Omron CX-Programmer project 新工程 (CX-Programmer 9.73)

# PLC LHJ_PLC: CQM1H CPU51
; 山东平度光明2003/08/20

## Global symbols (name address type ; comment)
0.00 BOOL  ; 上环升
0.00 BOOL  ; 上环升
0.01 BOOL  ; 上环降
0.01 BOOL  ; 上环降
0.02 BOOL  ; 下环升
0.02 BOOL  ; 下环升
0.03 BOOL  ; 下环降
0.03 BOOL  ; 下环降
0.04 BOOL  ; 支臂进
0.04 BOOL  ; 支臂进
0.05 BOOL  ; 支臂升
0.05 BOOL  ; 支臂升
0.06 BOOL  ; 定型
0.06 BOOL  ; 定型
0.07 BOOL  ; 合模
0.07 BOOL  ; 合模
0.08 BOOL  ; 开模
0.08 BOOL  ; 开模
0.09 BOOL  ; 急停
0.09 BOOL  ; 急停
0.10 BOOL  ; 机械手闭合
0.10 BOOL  ; 机械手闭合
0.11 BOOL  ; 机械手张开
0.11 BOOL  ; 机械手张开
0.12 BOOL  ; 转入
0.12 BOOL  ; 转入
0.13 BOOL  ; 机械手出
0.13 BOOL  ; 机械手出
0.14 BOOL  ; 机械手升
0.14 BOOL  ; 机械手升
0.15 BOOL  ; 机械手降
0.15 BOOL  ; 机械手降
100.00 BOOL  ; 上环升
100.00 BOOL  ; 上环升
100.01 BOOL  ; 上环降
100.01 BOOL  ; 上环降
100.02 BOOL  ; 下环升
100.02 BOOL  ; 下环升
100.03 BOOL  ; 下环降
100.03 BOOL  ; 下环降
100.04 BOOL  ; 支臂进
100.04 BOOL  ; 支臂进
100.05 BOOL  ; 支臂出
100.05 BOOL  ; 支臂出
100.06 BOOL  ; 支臂停
100.06 BOOL  ; 支臂停
100.07 BOOL  ; 支臂升
100.07 BOOL  ; 支臂升
100.08 BOOL  ; 油泵进
100.08 BOOL  ; 油泵进
100.09 BOOL  ; 油泵回
100.09 BOOL  ; 油泵回
100.10 BOOL  ; 合模换向
100.10 BOOL  ; 合模换向
100.11 BOOL  ; 开模换向
100.11 BOOL  ; 开模换向
100.12 BOOL  ; 抱闸
100.12 BOOL  ; 抱闸
100.13 BOOL  ; 合模
100.13 BOOL  ; 合模
100.14 BOOL  ; 开模
100.14 BOOL  ; 开模
101.00 BOOL  ; 定型
101.00 BOOL  ; 定型
101.01 BOOL  ; 二次定型
101.01 BOOL  ; 二次定型
101.02 BOOL  ; 左手闭合
101.02 BOOL  ; 左手闭合
101.03 BOOL  ; 右手闭合
101.03 BOOL  ; 右手闭合
101.04 BOOL  ; 左手降
101.04 BOOL  ; 左手降
101.05 BOOL  ; 右手降
101.05 BOOL  ; 右手降
101.06 BOOL  ; 左手停
101.06 BOOL  ; 左手停
101.07 BOOL  ; 右手停
101.07 BOOL  ; 右手停
101.08 BOOL  ; 左手入
101.08 BOOL  ; 左手入
101.09 BOOL  ; 右手入
101.09 BOOL  ; 右手入
101.10 BOOL  ; 左手出
101.10 BOOL  ; 左手出
101.11 BOOL  ; 右手出
101.11 BOOL  ; 右手出
101.12 BOOL  ; 自动指示灯
101.12 BOOL  ; 自动指示灯
101.13 BOOL  ; 硫化压力灯
101.14 BOOL  ; 硫化压力灯
101.14 BOOL  ; 硫化灯
101.15 BOOL  ; 硫化，延时硫化灯
101.15 BOOL  ; 硫化，延时硫化灯
102.00 BOOL  ; 内压蒸汽进
102.00 BOOL  ; 内压蒸汽进
102.01 BOOL  ; 内压蒸汽关
102.01 BOOL  ; 内压蒸汽关
102.02 BOOL  ; 二次水开
102.02 BOOL  ; 二次水开
102.03 BOOL  ; 二次水关
102.03 BOOL  ; 二次水关
102.04 BOOL  ; 热水回开
102.04 BOOL  ; 热水回开
102.05 BOOL  ; 热水回关
102.05 BOOL  ; 热水回关
102.06 BOOL  ; 5BAR热水回开
102.06 BOOL  ; 5BAR热水回开
102.07 BOOL  ; 5BAR热水回关
102.07 BOOL  ; 5BAR热水回关
102.08 BOOL  ; 0BAR热水回开
102.08 BOOL  ; 0BAR热水回开
102.09 BOOL  ; 0BAR热水回关
102.09 BOOL  ; 0BAR热水回关
102.10 BOOL  ; 抽真空开
102.11 BOOL  ; 抽真空关
102.12 BOOL  ; 外压（温）进开
102.13 BOOL  ; 外压（温）进关
102.14 BOOL  ; 冷水进回开
102.14 BOOL  ; 冷水进回开
102.15 BOOL  ; 冷水进回关
102.15 BOOL  ; 冷水进回关
103.00 BOOL  ; 外温进开
103.00 BOOL  ; 外温进开
103.01 BOOL  ; 活络模缩
103.02 BOOL  ; 活络模伸
103.02 BOOL  ; 活络模伸
103.03 BOOL  ; 活络模缩
103.03 BOOL  ; 活络模缩
103.04 BOOL  ; 挡胎杆降
103.04 BOOL  ; 挡胎杆降
103.05 BOOL  ; 活络模溢流
103.06 BOOL  ; 下环降停阀（有电通水）
103.08 BOOL  ; 报警灯
103.10 BOOL  ; 正常状态灯
103.12 BOOL  ; 程控气源失压报警
103.12 BOOL  ; 程控气源失压报警
104 CHANNEL  ; 外温回汽
104 CHANNEL  ; 外温回汽
105 CHANNEL  ; 进汽
105 CHANNEL  ; 进汽
11.10 BOOL  ; 左手转出
11.10 BOOL  ; 左手转出
13.15 BOOL  ; 延时硫化信号
13.15 BOOL  ; 延时硫化信号
14.00 BOOL  ; 实际压力大于设定的0.5公斤
14.00 BOOL  ; 实际压力大于设定的0.5公斤
15.00 BOOL  ; 备用
15.05 BOOL  ; 13.13
1.00 BOOL  ; 机械手停
1.00 BOOL  ; 机械手停
1.01 BOOL  ; 硫化延时
1.01 BOOL  ; 硫化延时
1.04 BOOL  ; 程序控制器
1.04 BOOL  ; 程序控制器
1.05 BOOL  ; 自动
1.05 BOOL  ; 自动
1.06 BOOL  ; 手动排
1.06 BOOL  ; 手动排
1.07 BOOL  ; 润滑
1.07 BOOL  ; 润滑
1.08 BOOL  ; 返回
1.08 BOOL  ; 返回
1.09 BOOL  ; 活络模升
1.09 BOOL  ; 活络模伸
1.10 BOOL  ; 活络模缩
1.10 BOOL  ; 活络模缩
1.11 BOOL  ; 挡胎杆升
1.13 BOOL  ; 机手（左）
1.13 BOOL  ; 机手（左）
1.14 BOOL  ; 机械手双
1.14 BOOL  ; 机械手双
1.15 BOOL  ; 机手（右）
1.15 BOOL  ; 机手（右）
22 CHANNEL  ; 动作序号
22.00 BOOL  ; 开模极限（编）
22.00 BOOL  ; 开模极限（编）
22.01 BOOL  ; 下环升
22.01 BOOL  ; 下环升
22.02 BOOL  ; 合模停（编）
22.02 BOOL  ; 合模停（编）
22.03 BOOL  ; 二次定型（编）
22.03 BOOL  ; 二次定型（编）
22.04 BOOL  ; 合模极限（编）
22.04 BOOL  ; 合模极限（编）
22.05 BOOL  ; 活络模伸（编）
22.05 BOOL  ; 活络模伸（编）
22.06 BOOL  ; 活络模缩（编）
22.06 BOOL  ; 活络模缩（编）
22.07 BOOL  ; 活络模保持
22.07 BOOL  ; 活络模保持
22 CHANNEL  ; 动作序号
233 CHANNEL  ; 热板温度采集
234 CHANNEL  ; 模套温度采集
236 CHANNEL  ; 模套温度电气转换器控制值
237 CHANNEL  ; 热板温度电气转换器控制值
23.00 BOOL  ; 达到设定步序
23.00 BOOL  ; 达到设定步序
26 CHANNEL  ; 判断步时间设定为0
26.00 BOOL  ; 第1步时间为0
26.00 BOOL  ; 第1步时间为0
26.01 BOOL  ; 第2步时间为0
26.01 BOOL  ; 第2步时间为0
26.02 BOOL  ; 第3步时间为0
26.02 BOOL  ; 第3步时间为0
26.03 BOOL  ; 第4步时间为0
26.03 BOOL  ; 第4步时间为0
26.04 BOOL  ; 第5步时间为0
26.04 BOOL  ; 第5步时间为0
26.05 BOOL  ; 第6步时间为0
26.05 BOOL  ; 第6步时间为0
26.06 BOOL  ; 第7步时间为0
26.06 BOOL  ; 第7步时间为0
26.07 BOOL  ; 8步时间为0
26.07 BOOL  ; 8步时间为0
26.08 BOOL  ; 九步时间为0
26.08 BOOL  ; 九步时间为0
26.09 BOOL  ; 第十步时间为0
26.09 BOOL  ; 第十步时间为0
26.10 BOOL  ; 11步时间为0
26.10 BOOL  ; 11步时间为0
26.11 BOOL  ; 12步时间为0
26.11 BOOL  ; 12步时间为0
26.12 BOOL  ; 第13步时间为0
26.12 BOOL  ; 第13步时间为0
26.13 BOOL  ; 第14步时间为0
26.13 BOOL  ; 第14步时间为0
26.14 BOOL  ; 第15步时间为0
26.14 BOOL  ; 第15步时间为0
26.15 BOOL  ; 第16步时间为0
26.15 BOOL  ; 第16步时间为0
26 CHANNEL  ; 判断步时间设定为0
2.00 BOOL  ; 抱闸
2.00 BOOL  ; 抱闸
2.01 BOOL  ; 内压
2.03 BOOL  ; 下环升
2.03 BOOL  ; 下环升
2.04 BOOL  ; 下环降
2.04 BOOL  ; 下环降
2.05 BOOL  ; 支臂进
2.05 BOOL  ; 支臂进
2.06 BOOL  ; 支臂停
2.06 BOOL  ; 支臂停
2.07 BOOL  ; 支臂降
2.07 BOOL  ; 支臂降
2.08 BOOL  ; 支臂出
2.08 BOOL  ; 支臂出
2.09 BOOL  ; 左手张开
2.09 BOOL  ; 左手张开
2.10 BOOL  ; 右手张开
2.10 BOOL  ; 右手张开
2.11 BOOL  ; 左手闭合
2.11 BOOL  ; 左手闭合
2.12 BOOL  ; 右手闭合
2.12 BOOL  ; 右手闭合
2.15 BOOL  ; 左手上限
2.15 BOOL  ; 左手上限
30.00 BOOL  ; 安全联锁
30.00 BOOL  ; 安全联锁
30.01 BOOL  ; 下环联锁
30.01 BOOL  ; 下环联锁
30.02 BOOL  ; 支臂联锁
30.02 BOOL  ; 支臂联锁
30.03 BOOL  ; 机手联锁
30.03 BOOL  ; 机手联锁
30.15 BOOL  ; 动作条件
30.15 BOOL  ; 动作条件
3.00 BOOL  ; 右手上限
3.00 BOOL  ; 右手上限
3.01 BOOL  ; 左手入
3.01 BOOL  ; 左手入
3.02 BOOL  ; 右手入
3.02 BOOL  ; 右手入
3.03 BOOL  ; 左手转出
3.03 BOOL  ; 左手转出
3.04 BOOL  ; 右手转出
3.04 BOOL  ; 右手转出
3.05 BOOL  ; 左手放胎
3.05 BOOL  ; 左手放胎
3.06 BOOL  ; 右手放胎
3.06 BOOL  ; 右手放胎
3.07 BOOL  ; 左手触胎
3.07 BOOL  ; 左手触胎
3.08 BOOL  ; 右手触胎
3.08 BOOL  ; 右手触胎
3.09 BOOL  ; 合模极限
3.09 BOOL  ; 合模极限
3.10 BOOL  ; 开模极限
3.10 BOOL  ; 开模极限
3.11 BOOL  ; 左安全开关
3.11 BOOL  ; 左安全开关
3.12 BOOL  ; 右安全开关
3.12 BOOL  ; 右安全开关
3.13 BOOL  ; 左活络模伸
3.13 BOOL  ; 左活络模伸
3.14 BOOL  ; 右活络模伸
3.14 BOOL  ; 右活络模伸
3.15 BOOL  ; 左活络模缩
3.15 BOOL  ; 左活络模缩
40.05 BOOL  ; 自动合模
40.05 BOOL  ; 自动合模
40.06 BOOL  ; 合模延时自锁
40.06 BOOL  ; 合模延时自锁
40.07 BOOL  ; 合模
40.07 BOOL  ; 合模
40.10 BOOL  ; 开模条件
40.10 BOOL  ; 开模条件
40.11 BOOL  ; 开模
40.11 BOOL  ; 开模
40.12 BOOL  ; 上环升条件1
40.12 BOOL  ; 上环升条件1
40.13 BOOL  ; 上环升条件1+2
40.13 BOOL  ; 上环升条件1+2
40.14 BOOL  ; 下环升条件
40.14 BOOL  ; 下环升条件
40.15 BOOL  ; 卸胎支臂停条件
40.15 BOOL  ; 卸胎支臂停条件
41.01 BOOL  ; 下环升
41.01 BOOL  ; 下环升
42.15 BOOL  ; 自动
42.15 BOOL  ; 自动
49.07 BOOL  ; 8-16步时间
49.07 BOOL  ; 8-16步时间
49.13 BOOL  ; 硫化结束步序清零
49.13 BOOL  ; 硫化结束步序清零
49.14 BOOL  ; 硫化结束
49.14 BOOL  ; 硫化结束
4.00 BOOL  ; 右活络模缩
4.00 BOOL  ; 右活络模缩
4.01 BOOL  ; 编码器输入1
4.01 BOOL  ; 编码器输入1
4.02 BOOL  ; 编码器输入2
4.02 BOOL  ; 编码器输入2
4.03 BOOL  ; 编码器输入3
4.03 BOOL  ; 编码器输入3
4.04 BOOL  ; 编码器输入4
4.04 BOOL  ; 编码器输入4
4.05 BOOL  ; 编码器输入5
4.05 BOOL  ; 编码器输入5
4.06 BOOL  ; 编码器输入6
4.06 BOOL  ; 编码器输入6
4.07 BOOL  ; 编码器输入7
4.07 BOOL  ; 编码器输入7
4.08 BOOL  ; 编码器输入8
4.08 BOOL  ; 编码器输入8
4.11 BOOL  ; 机械手切换
4.11 BOOL  ; 机械手切换
5 CHANNEL  ; 外温码
50.00 BOOL  ; 机械手转入自动
50.00 BOOL  ; 机械手转入自动
50.01 BOOL  ; 机械手转入自动
50.01 BOOL  ; 机械手转入自动
50.02 BOOL  ; 机手放胎条件
50.02 BOOL  ; 机手放胎条件
50.04 BOOL  ; 机手入自锁
50.04 BOOL  ; 机手入自锁
51.00 BOOL  ; 合模信号
51.00 BOOL  ; 合模信号
59.15 BOOL  ; 硫化条件
59.15 BOOL  ; 硫化条件
5 CHANNEL  ; 外温码
75.00 BOOL  ; 15步走完脉冲
75.00 BOOL  ; 15步走完脉冲
75.02 BOOL  ; 1步走完脉冲
75.02 BOOL  ; 1步走完脉冲
75.03 BOOL  ; 2步走完脉冲
75.03 BOOL  ; 2步走完脉冲
75.15 BOOL  ; 14步走完脉冲
75.15 BOOL  ; 14步走完脉冲
76.00 BOOL  ; 16步走完脉冲
76.00 BOOL  ; 16步走完脉冲
79.00 BOOL  ; 左闭合信号
79.00 BOOL  ; 左闭合信号
79.01 BOOL  ; 右闭信号
79.01 BOOL  ; 右闭信号
CNT001 BOOL  ; 初始化
CNT001 BOOL  ; 初始化
CNT002 BOOL  ; 第一步时间
CNT002 BOOL  ; 第一步时间
CNT003 BOOL  ; 第二步时间
CNT003 BOOL  ; 第二步时间
CNT004 BOOL  ; 第三步时间
CNT004 BOOL  ; 第三步时间
CNT005 BOOL  ; 第4步时间
CNT005 BOOL  ; 第4步时间
CNT006 BOOL  ; 第五步时间
CNT006 BOOL  ; 第五步时间
CNT007 BOOL  ; 第6步时间
CNT007 BOOL  ; 第6步时间
CNT008 BOOL  ; 第7步时间
CNT008 BOOL  ; 第7步时间
CNT009 BOOL  ; 第八步时
CNT009 BOOL  ; 第八步时
CNT010 BOOL  ; 第九步时
CNT010 BOOL  ; 第九步时
CNT011 BOOL  ; 第十步时
CNT011 BOOL  ; 第十步时
CNT012 BOOL  ; 第11步时间
CNT012 BOOL  ; 第11步时间
CNT013 BOOL  ; 第12步时间
CNT013 BOOL  ; 第12步时间
CNT014 BOOL  ; 第13步时间
CNT014 BOOL  ; 第13步时间
CNT015 BOOL  ; 第14步时间
CNT015 BOOL  ; 第14步时间
CNT016 BOOL  ; 第15步时间
CNT016 BOOL  ; 第15步时间
CNT017 BOOL  ; 第16步时间
CNT017 BOOL  ; 第16步时间
CNT018 BOOL  ; 硫化复位
CNT018 BOOL  ; 硫化复位
CNT022 BOOL  ; 延时硫化时间
CNT022 BOOL  ; 延时硫化时间
DM10 CHANNEL  ; 硫化总时间
DM1020 CHANNEL  ; PID模套温度设定二进值码
DM1021 CHANNEL  ; PID模套温度P参数
DM1026 CHANNEL  ; 模套温度PID的C+6
DM1055 CHANNEL  ; 模套温度PID控回汽
DM1055 CHANNEL  ; 温度PID控回汽
DM1060 CHANNEL  ; PID热板设定二进制码
DM1061 CHANNEL  ; PID热板P参数
DM1066 CHANNEL  ; 热板PID的C+6
DM1120 CHANNEL  ; 模套实际显示值
DM1122 CHANNEL  ; 内温实际显示值
DM1122 CHANNEL  ; 内温实际显示值
DM1126 CHANNEL  ; 内压实际显示值
DM1126 CHANNEL  ; 内压实际显示值
DM1128 CHANNEL  ; 实际热板温度显示值
DM1148 CHANNEL  ; 设定值加0.05公斤
DM1148 CHANNEL  ; 设定值加0.05公斤
DM1207 CHANNEL  ; 模套温度PID控制
DM1212 CHANNEL  ; 热板温度PID控制
DM1214 CHANNEL  ; 进汽阀开启度
DM1214 CHANNEL  ; 模套进汽阀开启度
DM1220 CHANNEL  ; 模套实际外温二进值码
DM1222 CHANNEL  ; 实际内温二进制码
DM1222 CHANNEL  ; 实际内温二进制码
DM1224 CHANNEL  ; 实际内压二进制码
DM1224 CHANNEL  ; 实际内压二进制码
DM1226 CHANNEL  ; 实际外压二进制码
DM1226 CHANNEL  ; 实际外压二进制码
DM1228 CHANNEL  ; PID热板实际温度二进值码
DM1230 CHANNEL  ; 实际内压MPa
DM1230 CHANNEL  ; 实际内压MPa
DM1232 CHANNEL  ; 实际外压MPa
DM1232 CHANNEL  ; 实际外压MPa
DM1238 CHANNEL  ; 压力低于设定值0.1公斤
DM1238 CHANNEL  ; 压力低于设定值0.1公斤
DM1242 CHANNEL  ; 热板进汽阀门开启度
DM170 CHANNEL  ; 模套温度设定值二进值码
DM172 CHANNEL  ; PPC热板温度设定值二进值码
DM400 CHANNEL  ; 步序一时间
DM400 CHANNEL  ; 步序一时间
DM401 CHANNEL  ; 步序二时间
DM401 CHANNEL  ; 步序二时间
DM402 CHANNEL  ; 步序三时间
DM402 CHANNEL  ; 步序三时间
DM403 CHANNEL  ; 步序四时间
DM403 CHANNEL  ; 步序四时间
DM404 CHANNEL  ; 步序五时间
DM404 CHANNEL  ; 步序五时间
DM405 CHANNEL  ; 步序六时间
DM405 CHANNEL  ; 步序六时间
DM406 CHANNEL  ; 步序七时间
DM406 CHANNEL  ; 步序七时间
DM407 CHANNEL  ; 第八步时间
DM407 CHANNEL  ; 第八步时间
DM408 CHANNEL  ; 第九步时间
DM408 CHANNEL  ; 第九步时间
DM409 CHANNEL  ; 第十步时间
DM409 CHANNEL  ; 第十步时间
DM410 CHANNEL  ; 第11步时间
DM410 CHANNEL  ; 第11步时间
DM411 CHANNEL  ; 第12步时间
DM411 CHANNEL  ; 第12步时间
DM412 CHANNEL  ; 第13步时间
DM412 CHANNEL  ; 第13步时间
DM413 CHANNEL  ; 第14步时间
DM413 CHANNEL  ; 第14步时间
DM414 CHANNEL  ; 第15步时间
DM414 CHANNEL  ; 第15步时间
DM415 CHANNEL  ; 第16步时间
DM415 CHANNEL  ; 第16步时间
DM416 CHANNEL  ; 第1步阀门状态
DM416 CHANNEL  ; 第1步阀门状态
DM417 CHANNEL  ; 第2步阀门状态
DM417 CHANNEL  ; 第2步阀门状态
DM418 CHANNEL  ; 第3步阀门状态
DM418 CHANNEL  ; 第3步阀门状态
DM419 CHANNEL  ; 第4步阀门状态
DM419 CHANNEL  ; 第4步阀门状态
DM420 CHANNEL  ; 第5步阀门状态
DM420 CHANNEL  ; 第5步阀门状态
DM421 CHANNEL  ; 第6步阀门状态
DM421 CHANNEL  ; 第6步阀门状态
DM422 CHANNEL  ; 第7步阀门状态
DM422 CHANNEL  ; 第7步阀门状态
DM423 CHANNEL  ; 第8步 阀门状态
DM423 CHANNEL  ; 第8步 阀门状态
DM424 CHANNEL  ; 第9步阀门状态
DM424 CHANNEL  ; 第9步阀门状态
DM425 CHANNEL  ; 第10步阀门状态
DM425 CHANNEL  ; 第10步阀门状态
DM426 CHANNEL  ; 第11步阀门状态
DM426 CHANNEL  ; 第11步阀门状态
DM427 CHANNEL  ; 第12步阀门状态
DM427 CHANNEL  ; 第12步阀门状态
DM428 CHANNEL  ; 第13步阀门状态
DM428 CHANNEL  ; 第13步阀门状态
DM429 CHANNEL  ; 第14步阀门状态
DM429 CHANNEL  ; 第14步阀门状态
DM430 CHANNEL  ; 第15步阀门状态
DM430 CHANNEL  ; 第15步阀门状态
DM431 CHANNEL  ; 第16步阀门状态
DM431 CHANNEL  ; 第16步阀门状态
DM448 CHANNEL  ; 模套设定值
DM449 CHANNEL  ; PPC写模套P参数
DM460 CHANNEL  ; PPC写热板温度设定值
DM461 CHANNEL  ; PPC写热板P参数
DM489 CHANNEL  ; 合模延时时间
DM489 CHANNEL  ; 合模延时时间
DM490 CHANNEL  ; 卸胎臂停延时
DM490 CHANNEL  ; 卸胎臂停延时
DM491 CHANNEL  ; 机械手闭合延时
DM491 CHANNEL  ; 机械手闭合延时
DM492 CHANNEL  ; 上环降延时
DM492 CHANNEL  ; 上环降延时
DM495 CHANNEL  ; 上环升延时
DM495 CHANNEL  ; 下环降延时
DM496 CHANNEL  ; 硫化延时时间
DM496 CHANNEL  ; 硫化延时时间
DM503 CHANNEL  ; 总步序设定
DM503 CHANNEL  ; 总步序设定
DM800 CHANNEL  ; 位置表比较
DM800 CHANNEL  ; 位置表比较
DM930 CHANNEL  ; PPC读PLC外温二进制数
DM930 CHANNEL  ; PPC读PLC外温二进制数
DM931 CHANNEL  ; PPC读PLC内温二进制数
DM931 CHANNEL  ; PPC读PLC内温二进制数
DM932 CHANNEL  ; PPC读PLC内压二进制数
DM932 CHANNEL  ; PPC读PLC内压二进制数
DM933 CHANNEL  ; PPC读PLC外压二进制数
DM933 CHANNEL  ; PPC读PLC外压二进制数
DM934 CHANNEL  ; 硫化总时间显示
DM934 CHANNEL  ; 硫化总时间显示
DM935 CHANNEL  ; 步序时间显示
DM935 CHANNEL  ; 步序时间显示
DM936 CHANNEL  ; PPC硫化延时显示
DM936 CHANNEL  ; PPC硫化延时显示
DM937 CHANNEL  ; 模套进汽阀开启度
DM937 CHANNEL  ; 进汽阀开启度
DM938 CHANNEL  ; 编码器值
DM938 CHANNEL  ; 编码器值
DM939 CHANNEL  ; 当前步序
DM939 CHANNEL  ; 当前步序
DM940 CHANNEL  ; 总剩余时间
DM940 CHANNEL  ; 总剩余时间
DM941 CHANNEL  ; 阀门状态
DM941 CHANNEL  ; 阀门状态
DM942 CHANNEL  ; 硫化状态标志
DM942 CHANNEL  ; 硫化状态标志
DM943 CHANNEL  ; PPC读00-01通道地址
DM943 CHANNEL  ; PPC读00-01通道地址
DM945 CHANNEL  ; PPC读PLC02-03通道地址
DM945 CHANNEL  ; PPC读PLC02-03通道地址
DM947 CHANNEL  ; PPC读100-103通道地址
DM947 CHANNEL  ; PPC读100-103通道地址
DM951 CHANNEL  ; PPC热板进汽阀门开启度
HR31.00 BOOL  ; 自动硫化保护
HR31.00 BOOL  ; 自动硫化保护
TIM000 BOOL  ; 合模延时时间
TIM000 BOOL  ; 合模延时时间
TIM052 BOOL  ; 下环降延时
TIM052 BOOL  ; 下环降延时
TIM053 BOOL  ; 卸胎支臂停延时
TIM053 BOOL  ; 卸胎支臂停延时
TIM054 BOOL  ; 上环降延时
TIM054 BOOL  ; 上环降延时
TIM056 BOOL  ; 返回时间
TIM056 BOOL  ; 返回时间
TIM057 BOOL  ; 润滑时间
TIM057 BOOL  ; 润滑时间
TIM069 BOOL  ; 支臂降延时
TIM069 BOOL  ; 支臂降延时
TIM070 BOOL  ; 定型延时
TIM070 BOOL  ; 机械手闭合延时
TIM071 BOOL  ; 左手在外抓胎延时
TIM071 BOOL  ; 左手在外抓胎延时
TIM072 BOOL  ; 右手在外抓胎延时
TIM072 BOOL  ; 右手在外抓胎延时
TIM079 BOOL  ; 内压
TIM079 BOOL  ; 内压

## Program 新程序1 (no task)
; 系统使用欧姆龙PLC CQM1H CPU51，通过编码器、温度传感器、压力传感器、机械手、阀门和安全开关等设备实现硫化过程的自动化控制。 / 系统只有在急停未触发且安全门关闭时，硫化流程才会启动，否则所有动作如合模和开模立即停止，确保操作安全。 / 硫化过程温度控制通过PID算法实现，利用PID模套温度设定值和PID热板温度设定值调整模套温度控制值和热板温度控制值，使温度稳定在设定值的±5%以内，确保硫化质量。 / 压力则通过内压蒸汽进和内压蒸汽关调节，保持在设定值的±0.5巴范围内，避免压力波动影响轮胎成型。 / 机械手动作由左手闭合、右手闭合、左手入、右手入等信号驱动，且左手闭合和右手闭合不会同时激活，且只能在编码器确认的安全区域内执行，防止机械冲突和越界。 / 硫化结束后，计时器触发复位，自动指示灯和硫化灯显示运行状态，系统准备下一轮操作。 / sn:3911-5900-9079-9900

### Section 段1

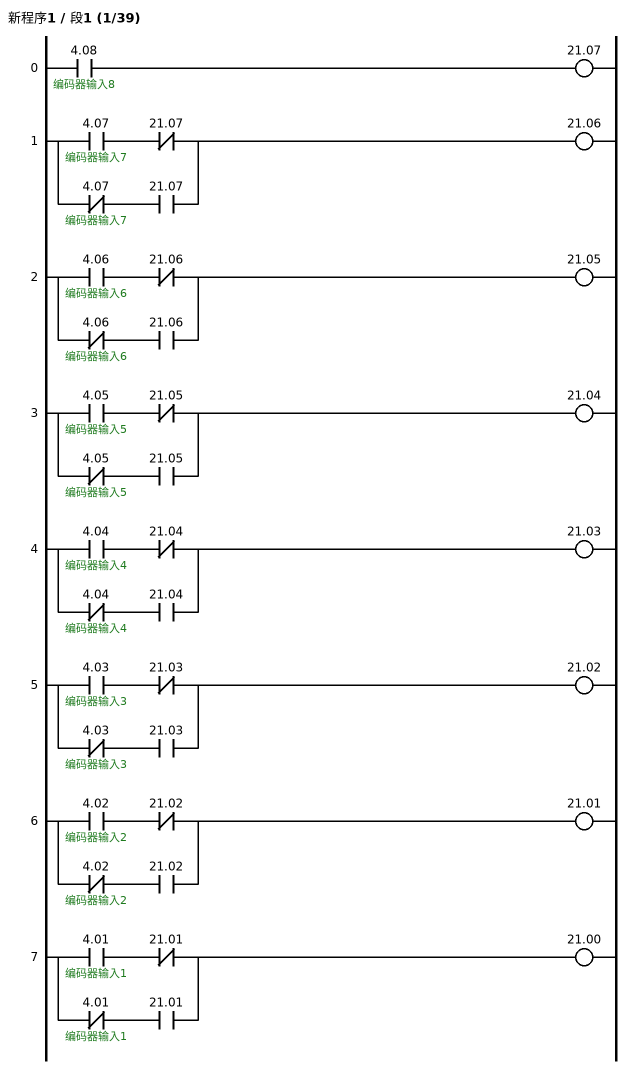
; rung 0
LD 4.08  ; 编码器输入8
OUT 21.07
; rung 1
LD 4.07  ; 编码器输入7
ANDNOT 21.07
LDNOT 4.07  ; 编码器输入7
AND 21.07
ORLD
OUT 21.06
; rung 2
LD 4.06  ; 编码器输入6
ANDNOT 21.06
LDNOT 4.06  ; 编码器输入6
AND 21.06
ORLD
OUT 21.05
; rung 3
LD 4.05  ; 编码器输入5
ANDNOT 21.05
LDNOT 4.05  ; 编码器输入5
AND 21.05
ORLD
OUT 21.04
; rung 4
LD 4.04  ; 编码器输入4
ANDNOT 21.04
LDNOT 4.04  ; 编码器输入4
AND 21.04
ORLD
OUT 21.03
; rung 5
LD 4.03  ; 编码器输入3
ANDNOT 21.03
LDNOT 4.03  ; 编码器输入3
AND 21.03
ORLD
OUT 21.02
; rung 6
LD 4.02  ; 编码器输入2
ANDNOT 21.02
LDNOT 4.02  ; 编码器输入2
AND 21.02
ORLD
OUT 21.01
; rung 7
LD 4.01  ; 编码器输入1
ANDNOT 21.01
LDNOT 4.01  ; 编码器输入1
AND 21.01
ORLD
OUT 21.00

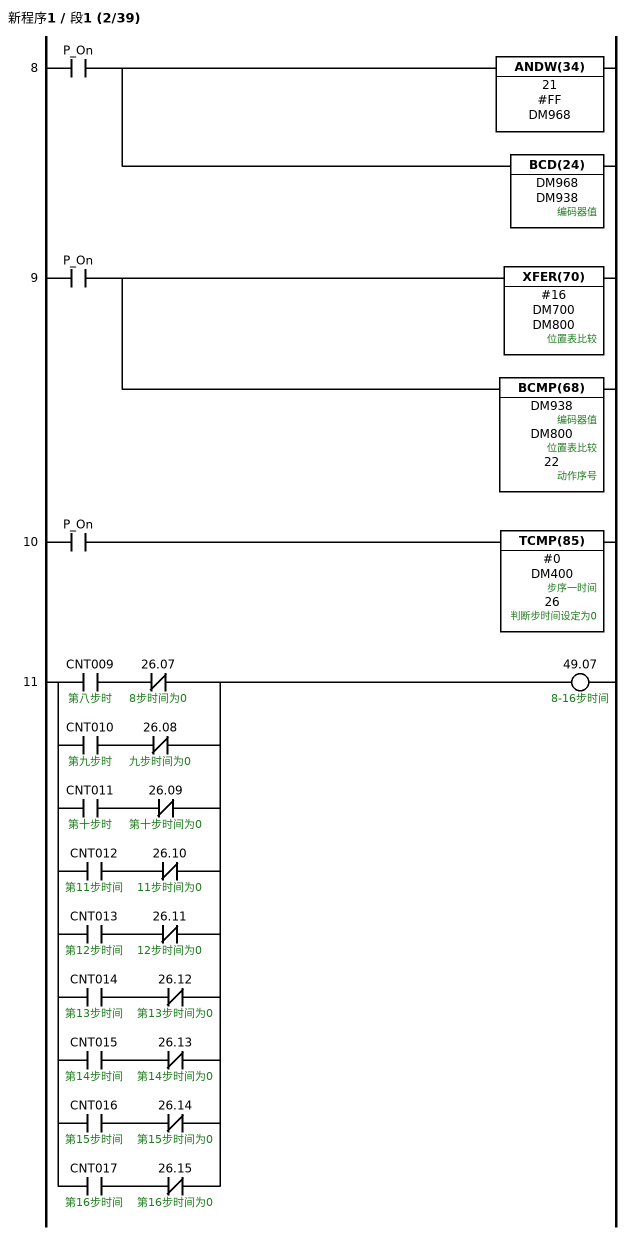
; rung 8
LD P_On
ANDW(34) 21 #FF DM968
BCD(24) DM968 DM938  ; 编码器值
; rung 9
LD P_On
XFER(70) #16 DM700 DM800  ; 位置表比较
BCMP(68) DM938 DM800 22  ; 编码器值, 位置表比较, 动作序号
; rung 10
LD P_On
TCMP(85) #0 DM400 26  ; 步序一时间, 判断步时间设定为0
; rung 11
LD CNT009  ; 第八步时
ANDNOT 26.07  ; 8步时间为0
LD CNT010  ; 第九步时
ANDNOT 26.08  ; 九步时间为0
ORLD
LD CNT011  ; 第十步时
ANDNOT 26.09  ; 第十步时间为0
ORLD
LD CNT012  ; 第11步时间
ANDNOT 26.10  ; 11步时间为0
ORLD
LD CNT013  ; 第12步时间
ANDNOT 26.11  ; 12步时间为0
ORLD
LD CNT014  ; 第13步时间
ANDNOT 26.12  ; 第13步时间为0
ORLD
LD CNT015  ; 第14步时间
ANDNOT 26.13  ; 第14步时间为0
ORLD
LD CNT016  ; 第15步时间
ANDNOT 26.14  ; 第15步时间为0
ORLD
LD CNT017  ; 第16步时间
ANDNOT 26.15  ; 第16步时间为0
ORLD
OUT 49.07  ; 8-16步时间

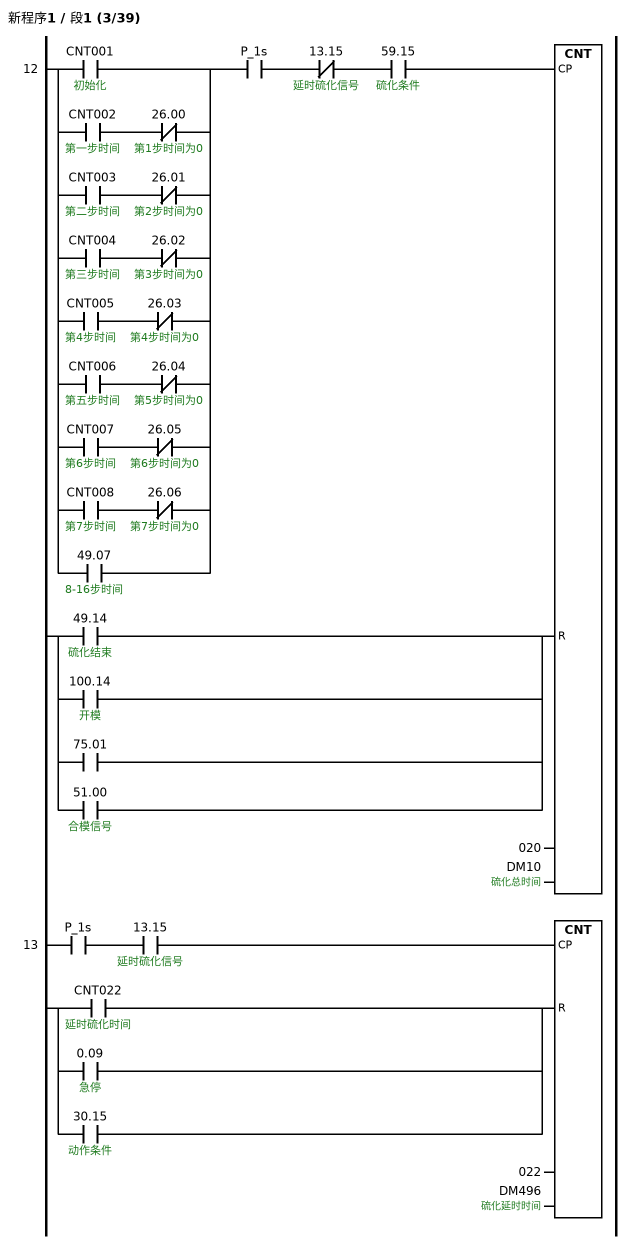
; rung 12
LD CNT001  ; 初始化
LD CNT002  ; 第一步时间
ANDNOT 26.00  ; 第1步时间为0
ORLD
LD CNT003  ; 第二步时间
ANDNOT 26.01  ; 第2步时间为0
ORLD
LD CNT004  ; 第三步时间
ANDNOT 26.02  ; 第3步时间为0
ORLD
LD CNT005  ; 第4步时间
ANDNOT 26.03  ; 第4步时间为0
ORLD
LD CNT006  ; 第五步时间
ANDNOT 26.04  ; 第5步时间为0
ORLD
LD CNT007  ; 第6步时间
ANDNOT 26.05  ; 第6步时间为0
ORLD
LD CNT008  ; 第7步时间
ANDNOT 26.06  ; 第7步时间为0
ORLD
OR 49.07  ; 8-16步时间
AND P_1s
ANDNOT 13.15  ; 延时硫化信号
AND 59.15  ; 硫化条件
LD 49.14  ; 硫化结束
OR 100.14  ; 开模
OR 75.01
OR 51.00  ; 合模信号
CNT 020 DM10  ; 硫化总时间
; rung 13
LD P_1s
AND 13.15  ; 延时硫化信号
LD CNT022  ; 延时硫化时间
OR 0.09  ; 急停
OR 30.15  ; 动作条件
CNT 022 DM496  ; 硫化延时时间

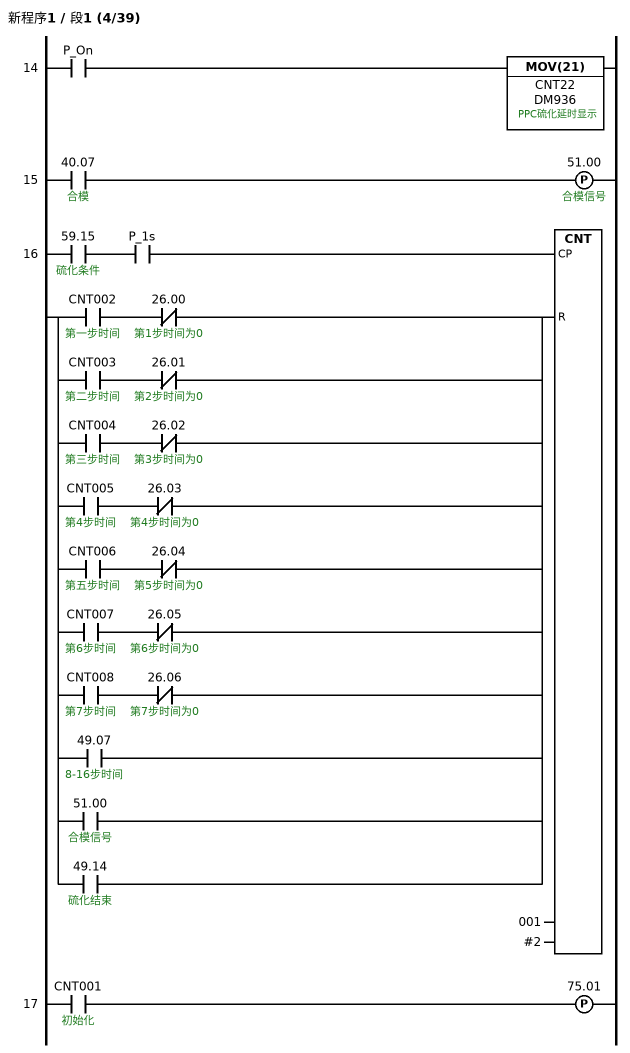
; rung 14
LD P_On
MOV(21) CNT22 DM936  ; PPC硫化延时显示
; rung 15
LD 40.07  ; 合模
DIFU(13) 51.00  ; 合模信号
; rung 16
LD 59.15  ; 硫化条件
AND P_1s
LD CNT002  ; 第一步时间
ANDNOT 26.00  ; 第1步时间为0
LD CNT003  ; 第二步时间
ANDNOT 26.01  ; 第2步时间为0
ORLD
LD CNT004  ; 第三步时间
ANDNOT 26.02  ; 第3步时间为0
ORLD
LD CNT005  ; 第4步时间
ANDNOT 26.03  ; 第4步时间为0
ORLD
LD CNT006  ; 第五步时间
ANDNOT 26.04  ; 第5步时间为0
ORLD
LD CNT007  ; 第6步时间
ANDNOT 26.05  ; 第6步时间为0
ORLD
LD CNT008  ; 第7步时间
ANDNOT 26.06  ; 第7步时间为0
ORLD
OR 49.07  ; 8-16步时间
OR 51.00  ; 合模信号
OR 49.14  ; 硫化结束
CNT 001 #2
; rung 17
LD CNT001  ; 初始化
DIFU(13) 75.01

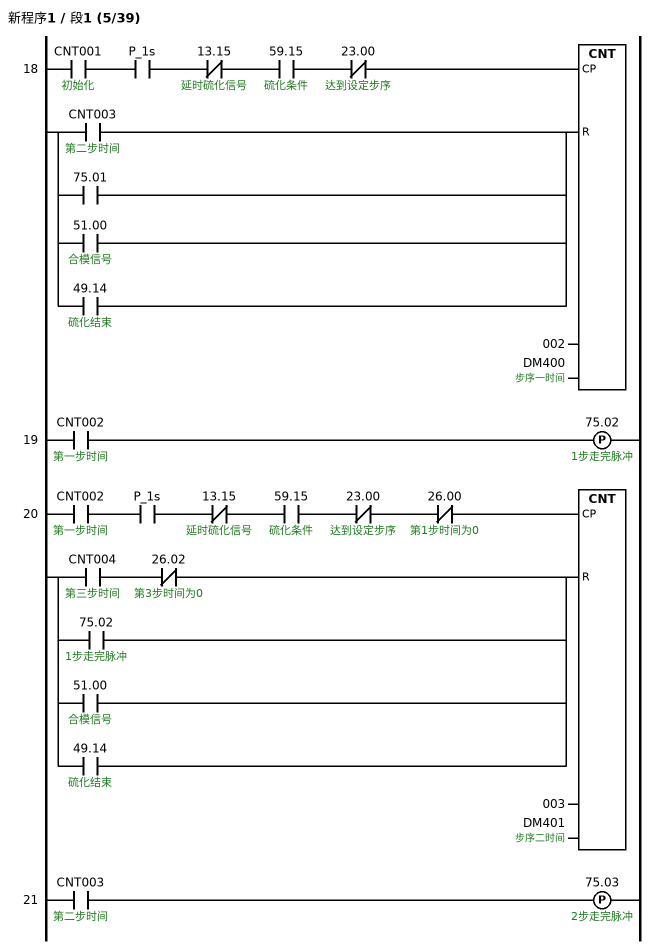
; rung 18
LD CNT001  ; 初始化
AND P_1s
ANDNOT 13.15  ; 延时硫化信号
AND 59.15  ; 硫化条件
ANDNOT 23.00  ; 达到设定步序
LD CNT003  ; 第二步时间
OR 75.01
OR 51.00  ; 合模信号
OR 49.14  ; 硫化结束
CNT 002 DM400  ; 步序一时间
; rung 19
LD CNT002  ; 第一步时间
DIFU(13) 75.02  ; 1步走完脉冲
; rung 20
LD CNT002  ; 第一步时间
AND P_1s
ANDNOT 13.15  ; 延时硫化信号
AND 59.15  ; 硫化条件
ANDNOT 23.00  ; 达到设定步序
ANDNOT 26.00  ; 第1步时间为0
LD CNT004  ; 第三步时间
ANDNOT 26.02  ; 第3步时间为0
OR 75.02  ; 1步走完脉冲
OR 51.00  ; 合模信号
OR 49.14  ; 硫化结束
CNT 003 DM401  ; 步序二时间
; rung 21
LD CNT003  ; 第二步时间
DIFU(13) 75.03  ; 2步走完脉冲

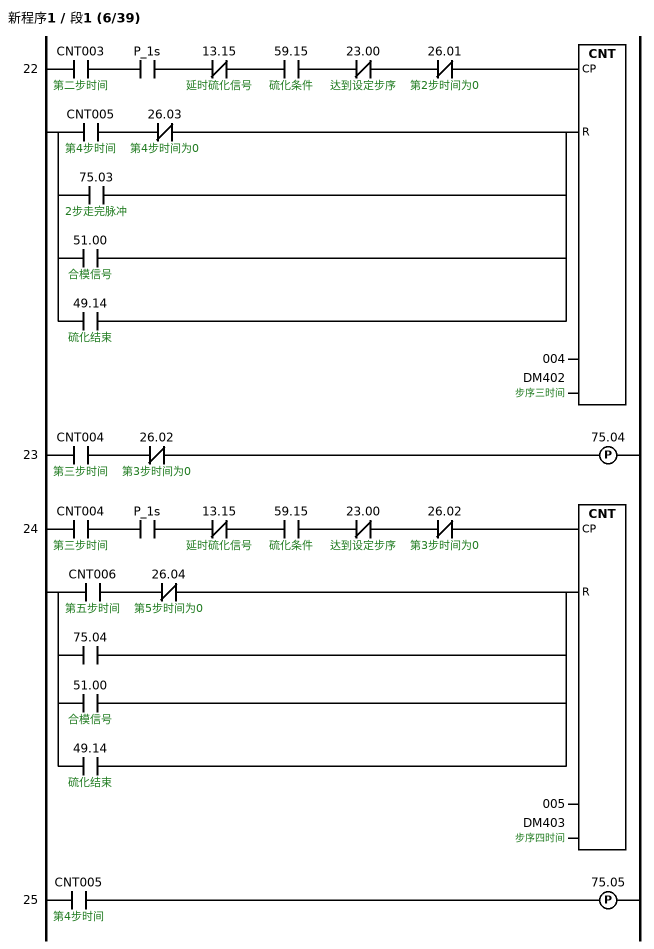
; rung 22
LD CNT003  ; 第二步时间
AND P_1s
ANDNOT 13.15  ; 延时硫化信号
AND 59.15  ; 硫化条件
ANDNOT 23.00  ; 达到设定步序
ANDNOT 26.01  ; 第2步时间为0
LD CNT005  ; 第4步时间
ANDNOT 26.03  ; 第4步时间为0
OR 75.03  ; 2步走完脉冲
OR 51.00  ; 合模信号
OR 49.14  ; 硫化结束
CNT 004 DM402  ; 步序三时间
; rung 23
LD CNT004  ; 第三步时间
ANDNOT 26.02  ; 第3步时间为0
DIFU(13) 75.04
; rung 24
LD CNT004  ; 第三步时间
AND P_1s
ANDNOT 13.15  ; 延时硫化信号
AND 59.15  ; 硫化条件
ANDNOT 23.00  ; 达到设定步序
ANDNOT 26.02  ; 第3步时间为0
LD CNT006  ; 第五步时间
ANDNOT 26.04  ; 第5步时间为0
OR 75.04
OR 51.00  ; 合模信号
OR 49.14  ; 硫化结束
CNT 005 DM403  ; 步序四时间
; rung 25
LD CNT005  ; 第4步时间
DIFU(13) 75.05

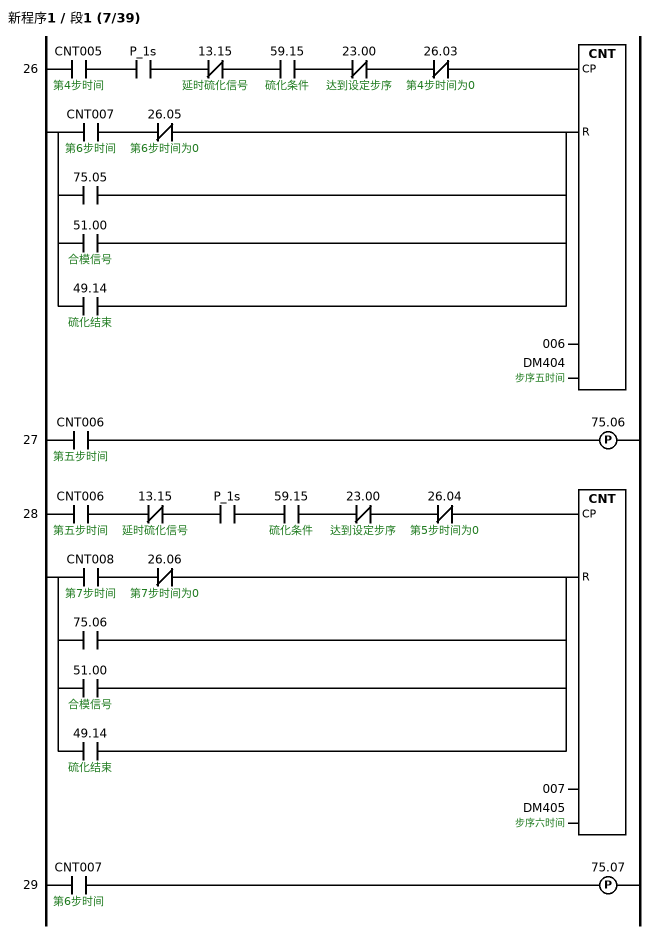
; rung 26
LD CNT005  ; 第4步时间
AND P_1s
ANDNOT 13.15  ; 延时硫化信号
AND 59.15  ; 硫化条件
ANDNOT 23.00  ; 达到设定步序
ANDNOT 26.03  ; 第4步时间为0
LD CNT007  ; 第6步时间
ANDNOT 26.05  ; 第6步时间为0
OR 75.05
OR 51.00  ; 合模信号
OR 49.14  ; 硫化结束
CNT 006 DM404  ; 步序五时间
; rung 27
LD CNT006  ; 第五步时间
DIFU(13) 75.06
; rung 28
LD CNT006  ; 第五步时间
ANDNOT 13.15  ; 延时硫化信号
AND P_1s
AND 59.15  ; 硫化条件
ANDNOT 23.00  ; 达到设定步序
ANDNOT 26.04  ; 第5步时间为0
LD CNT008  ; 第7步时间
ANDNOT 26.06  ; 第7步时间为0
OR 75.06
OR 51.00  ; 合模信号
OR 49.14  ; 硫化结束
CNT 007 DM405  ; 步序六时间
; rung 29
LD CNT007  ; 第6步时间
DIFU(13) 75.07

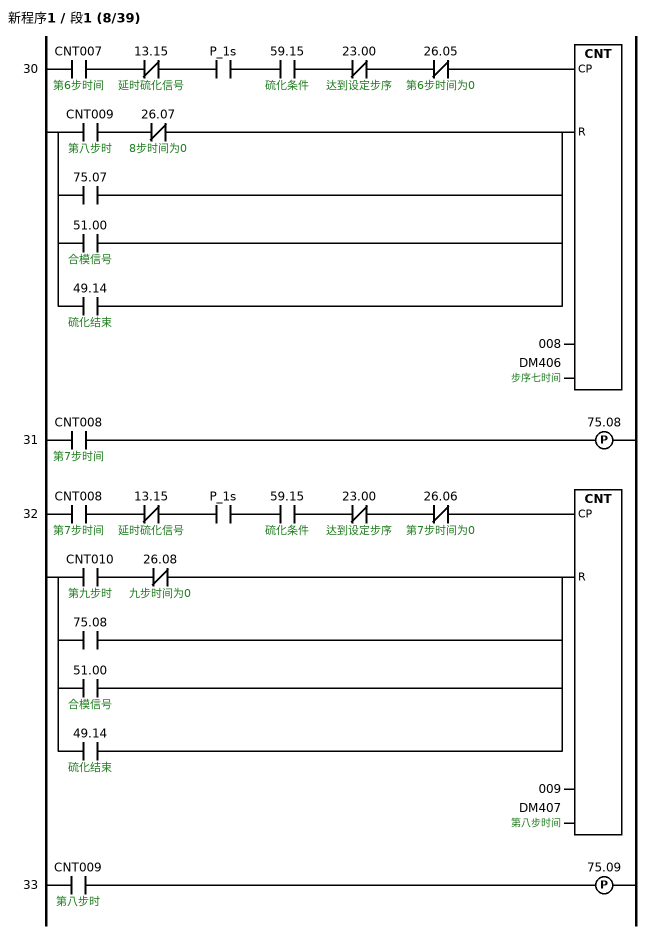
; rung 30
LD CNT007  ; 第6步时间
ANDNOT 13.15  ; 延时硫化信号
AND P_1s
AND 59.15  ; 硫化条件
ANDNOT 23.00  ; 达到设定步序
ANDNOT 26.05  ; 第6步时间为0
LD CNT009  ; 第八步时
ANDNOT 26.07  ; 8步时间为0
OR 75.07
OR 51.00  ; 合模信号
OR 49.14  ; 硫化结束
CNT 008 DM406  ; 步序七时间
; rung 31
LD CNT008  ; 第7步时间
DIFU(13) 75.08
; rung 32
LD CNT008  ; 第7步时间
ANDNOT 13.15  ; 延时硫化信号
AND P_1s
AND 59.15  ; 硫化条件
ANDNOT 23.00  ; 达到设定步序
ANDNOT 26.06  ; 第7步时间为0
LD CNT010  ; 第九步时
ANDNOT 26.08  ; 九步时间为0
OR 75.08
OR 51.00  ; 合模信号
OR 49.14  ; 硫化结束
CNT 009 DM407  ; 第八步时间
; rung 33
LD CNT009  ; 第八步时
DIFU(13) 75.09

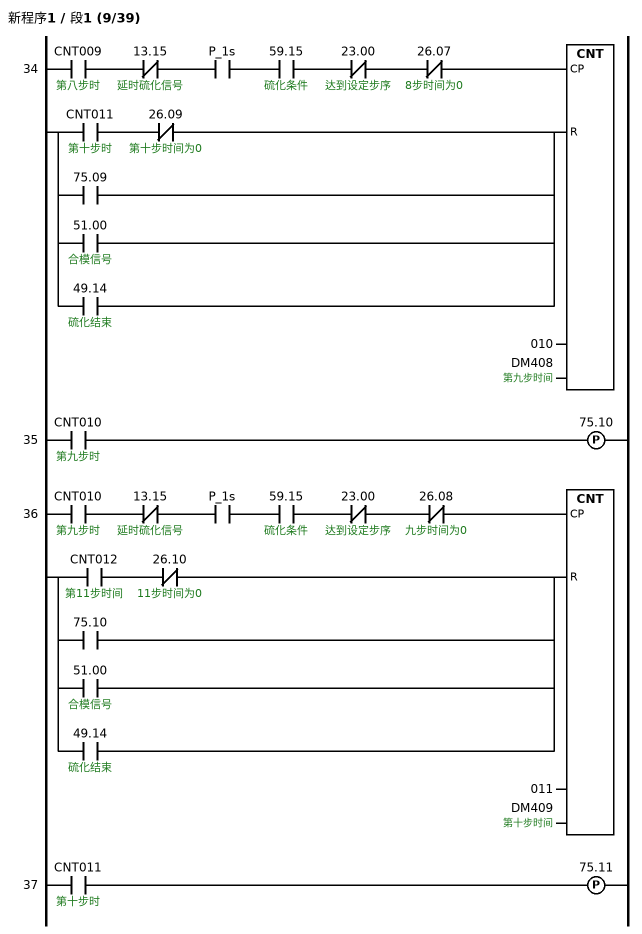
; rung 34
LD CNT009  ; 第八步时
ANDNOT 13.15  ; 延时硫化信号
AND P_1s
AND 59.15  ; 硫化条件
ANDNOT 23.00  ; 达到设定步序
ANDNOT 26.07  ; 8步时间为0
LD CNT011  ; 第十步时
ANDNOT 26.09  ; 第十步时间为0
OR 75.09
OR 51.00  ; 合模信号
OR 49.14  ; 硫化结束
CNT 010 DM408  ; 第九步时间
; rung 35
LD CNT010  ; 第九步时
DIFU(13) 75.10
; rung 36
LD CNT010  ; 第九步时
ANDNOT 13.15  ; 延时硫化信号
AND P_1s
AND 59.15  ; 硫化条件
ANDNOT 23.00  ; 达到设定步序
ANDNOT 26.08  ; 九步时间为0
LD CNT012  ; 第11步时间
ANDNOT 26.10  ; 11步时间为0
OR 75.10
OR 51.00  ; 合模信号
OR 49.14  ; 硫化结束
CNT 011 DM409  ; 第十步时间
; rung 37
LD CNT011  ; 第十步时
DIFU(13) 75.11

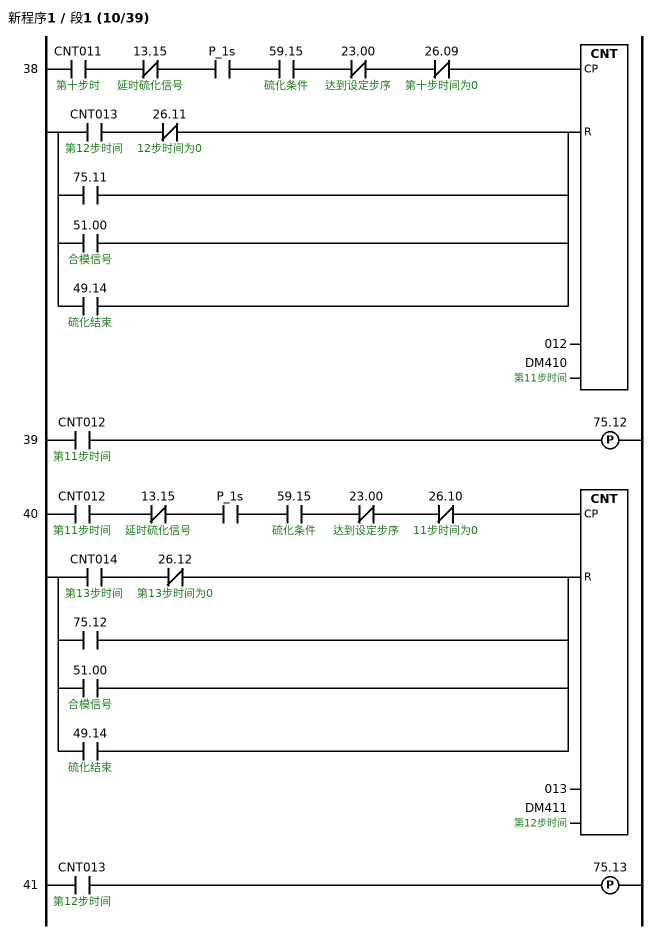
; rung 38
LD CNT011  ; 第十步时
ANDNOT 13.15  ; 延时硫化信号
AND P_1s
AND 59.15  ; 硫化条件
ANDNOT 23.00  ; 达到设定步序
ANDNOT 26.09  ; 第十步时间为0
LD CNT013  ; 第12步时间
ANDNOT 26.11  ; 12步时间为0
OR 75.11
OR 51.00  ; 合模信号
OR 49.14  ; 硫化结束
CNT 012 DM410  ; 第11步时间
; rung 39
LD CNT012  ; 第11步时间
DIFU(13) 75.12
; rung 40
LD CNT012  ; 第11步时间
ANDNOT 13.15  ; 延时硫化信号
AND P_1s
AND 59.15  ; 硫化条件
ANDNOT 23.00  ; 达到设定步序
ANDNOT 26.10  ; 11步时间为0
LD CNT014  ; 第13步时间
ANDNOT 26.12  ; 第13步时间为0
OR 75.12
OR 51.00  ; 合模信号
OR 49.14  ; 硫化结束
CNT 013 DM411  ; 第12步时间
; rung 41
LD CNT013  ; 第12步时间
DIFU(13) 75.13

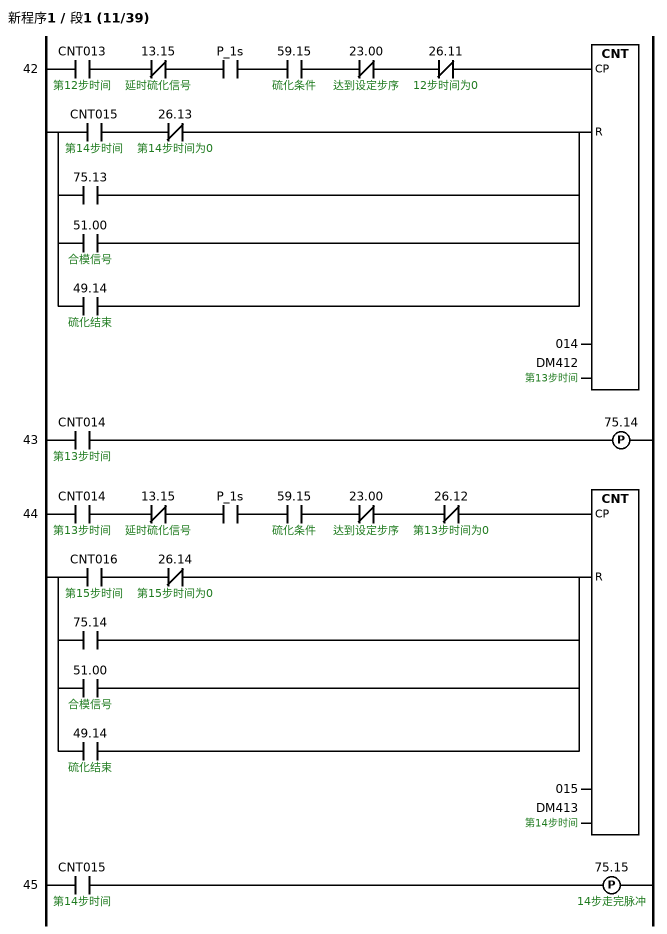
; rung 42
LD CNT013  ; 第12步时间
ANDNOT 13.15  ; 延时硫化信号
AND P_1s
AND 59.15  ; 硫化条件
ANDNOT 23.00  ; 达到设定步序
ANDNOT 26.11  ; 12步时间为0
LD CNT015  ; 第14步时间
ANDNOT 26.13  ; 第14步时间为0
OR 75.13
OR 51.00  ; 合模信号
OR 49.14  ; 硫化结束
CNT 014 DM412  ; 第13步时间
; rung 43
LD CNT014  ; 第13步时间
DIFU(13) 75.14
; rung 44
LD CNT014  ; 第13步时间
ANDNOT 13.15  ; 延时硫化信号
AND P_1s
AND 59.15  ; 硫化条件
ANDNOT 23.00  ; 达到设定步序
ANDNOT 26.12  ; 第13步时间为0
LD CNT016  ; 第15步时间
ANDNOT 26.14  ; 第15步时间为0
OR 75.14
OR 51.00  ; 合模信号
OR 49.14  ; 硫化结束
CNT 015 DM413  ; 第14步时间
; rung 45
LD CNT015  ; 第14步时间
DIFU(13) 75.15  ; 14步走完脉冲

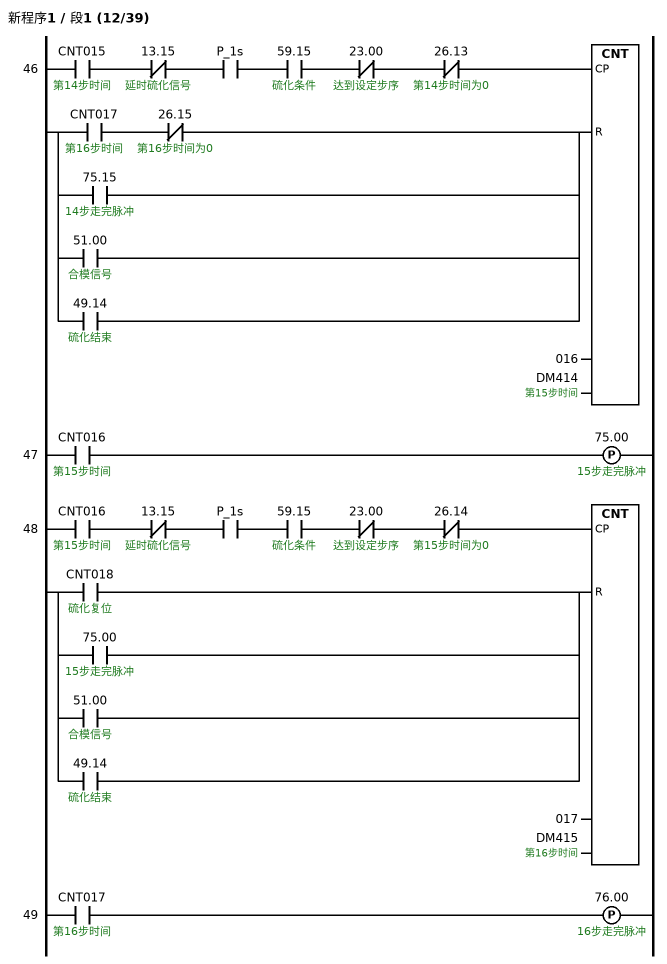
; rung 46
LD CNT015  ; 第14步时间
ANDNOT 13.15  ; 延时硫化信号
AND P_1s
AND 59.15  ; 硫化条件
ANDNOT 23.00  ; 达到设定步序
ANDNOT 26.13  ; 第14步时间为0
LD CNT017  ; 第16步时间
ANDNOT 26.15  ; 第16步时间为0
OR 75.15  ; 14步走完脉冲
OR 51.00  ; 合模信号
OR 49.14  ; 硫化结束
CNT 016 DM414  ; 第15步时间
; rung 47
LD CNT016  ; 第15步时间
DIFU(13) 75.00  ; 15步走完脉冲
; rung 48
LD CNT016  ; 第15步时间
ANDNOT 13.15  ; 延时硫化信号
AND P_1s
AND 59.15  ; 硫化条件
ANDNOT 23.00  ; 达到设定步序
ANDNOT 26.14  ; 第15步时间为0
LD CNT018  ; 硫化复位
OR 75.00  ; 15步走完脉冲
OR 51.00  ; 合模信号
OR 49.14  ; 硫化结束
CNT 017 DM415  ; 第16步时间
; rung 49
LD CNT017  ; 第16步时间
DIFU(13) 76.00  ; 16步走完脉冲

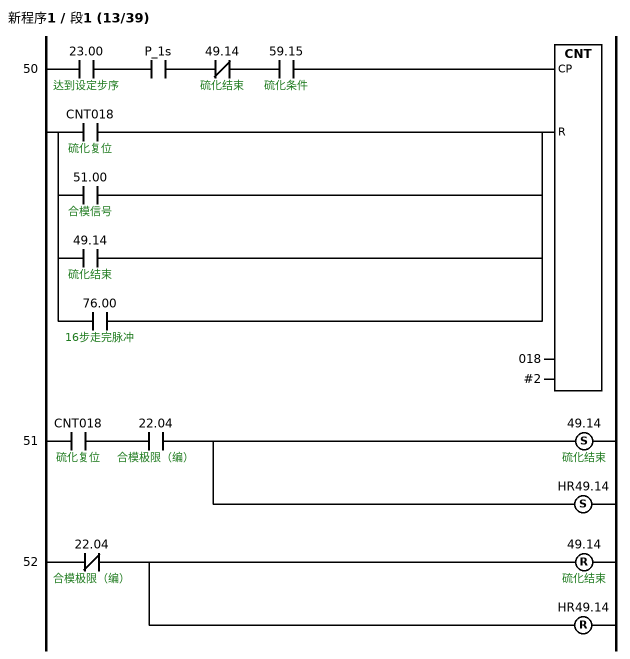
; rung 50
LD 23.00  ; 达到设定步序
AND P_1s
ANDNOT 49.14  ; 硫化结束
AND 59.15  ; 硫化条件
LD CNT018  ; 硫化复位
OR 51.00  ; 合模信号
OR 49.14  ; 硫化结束
OR 76.00  ; 16步走完脉冲
CNT 018 #2
; rung 51
LD CNT018  ; 硫化复位
AND 22.04  ; 合模极限（编）
SET 49.14  ; 硫化结束
SET HR49.14
; rung 52
LDNOT 22.04  ; 合模极限（编）
RSET 49.14  ; 硫化结束
RSET HR49.14

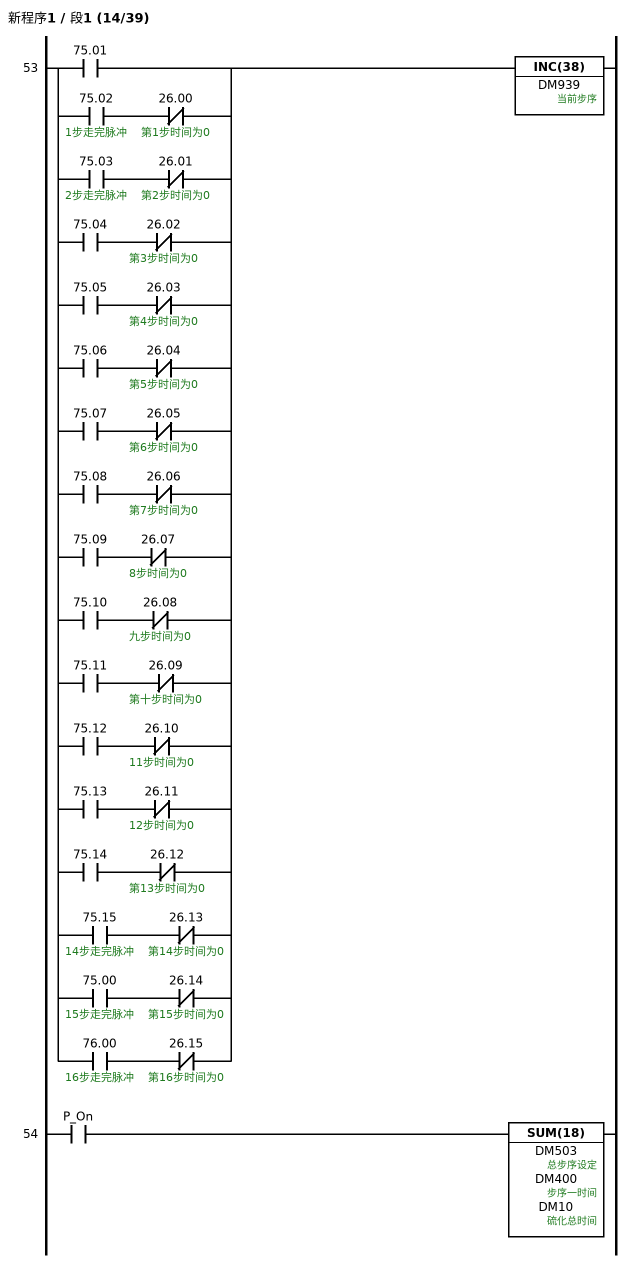
; rung 53
LD 75.01
LD 75.02  ; 1步走完脉冲
ANDNOT 26.00  ; 第1步时间为0
ORLD
LD 75.03  ; 2步走完脉冲
ANDNOT 26.01  ; 第2步时间为0
ORLD
LD 75.04
ANDNOT 26.02  ; 第3步时间为0
ORLD
LD 75.05
ANDNOT 26.03  ; 第4步时间为0
ORLD
LD 75.06
ANDNOT 26.04  ; 第5步时间为0
ORLD
LD 75.07
ANDNOT 26.05  ; 第6步时间为0
ORLD
LD 75.08
ANDNOT 26.06  ; 第7步时间为0
ORLD
LD 75.09
ANDNOT 26.07  ; 8步时间为0
ORLD
LD 75.10
ANDNOT 26.08  ; 九步时间为0
ORLD
LD 75.11
ANDNOT 26.09  ; 第十步时间为0
ORLD
LD 75.12
ANDNOT 26.10  ; 11步时间为0
ORLD
LD 75.13
ANDNOT 26.11  ; 12步时间为0
ORLD
LD 75.14
ANDNOT 26.12  ; 第13步时间为0
ORLD
LD 75.15  ; 14步走完脉冲
ANDNOT 26.13  ; 第14步时间为0
ORLD
LD 75.00  ; 15步走完脉冲
ANDNOT 26.14  ; 第15步时间为0
ORLD
LD 76.00  ; 16步走完脉冲
ANDNOT 26.15  ; 第16步时间为0
ORLD
INC(38) DM939  ; 当前步序
; rung 54
LD P_On
SUM(18) DM503 DM400 DM10  ; 总步序设定, 步序一时间, 硫化总时间

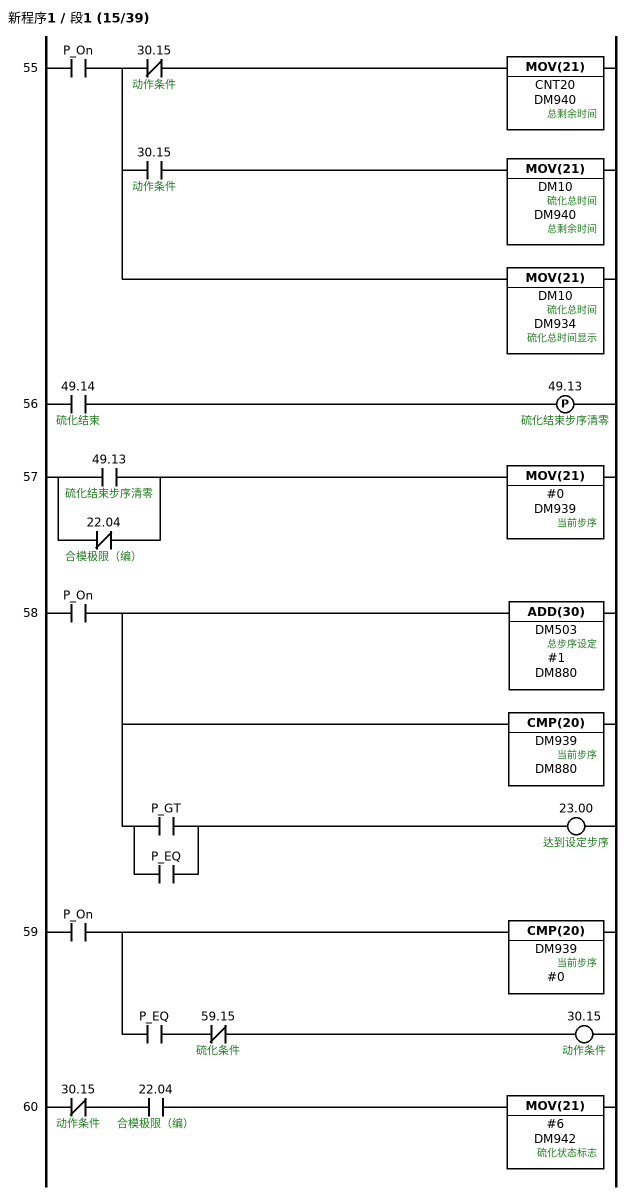
; rung 55
LD P_On
OUT TR0
ANDNOT 30.15  ; 动作条件
MOV(21) CNT20 DM940  ; 总剩余时间
LD TR0
AND 30.15  ; 动作条件
MOV(21) DM10 DM940  ; 硫化总时间, 总剩余时间
LD TR0
MOV(21) DM10 DM934  ; 硫化总时间, 硫化总时间显示
; rung 56
LD 49.14  ; 硫化结束
DIFU(13) 49.13  ; 硫化结束步序清零
; rung 57
LD 49.13  ; 硫化结束步序清零
ORNOT 22.04  ; 合模极限（编）
MOV(21) #0 DM939  ; 当前步序
; rung 58
LD P_On
ADD(30) DM503 #1 DM880  ; 总步序设定
CMP(20) DM939 DM880  ; 当前步序
LD P_GT
OR P_EQ
ANDLD
OUT 23.00  ; 达到设定步序
; rung 59
LD P_On
CMP(20) DM939 #0  ; 当前步序
AND P_EQ
ANDNOT 59.15  ; 硫化条件
OUT 30.15  ; 动作条件
; rung 60
LDNOT 30.15  ; 动作条件
AND 22.04  ; 合模极限（编）
MOV(21) #6 DM942  ; 硫化状态标志

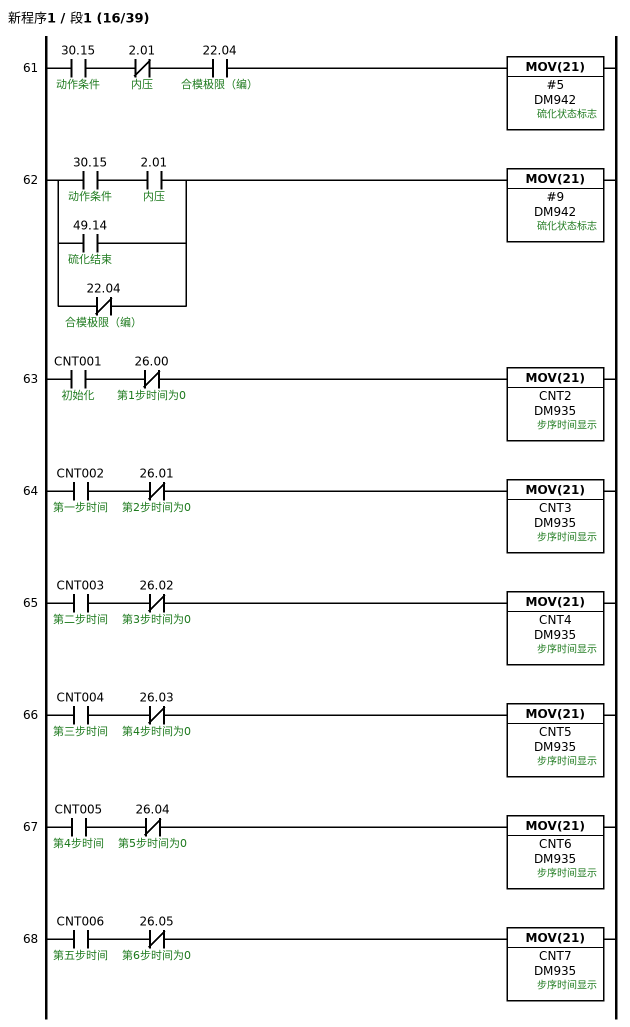
; rung 61
LD 30.15  ; 动作条件
ANDNOT 2.01  ; 内压
AND 22.04  ; 合模极限（编）
MOV(21) #5 DM942  ; 硫化状态标志
; rung 62
LD 30.15  ; 动作条件
AND 2.01  ; 内压
OR 49.14  ; 硫化结束
ORNOT 22.04  ; 合模极限（编）
MOV(21) #9 DM942  ; 硫化状态标志
; rung 63
LD CNT001  ; 初始化
ANDNOT 26.00  ; 第1步时间为0
MOV(21) CNT2 DM935  ; 步序时间显示
; rung 64
LD CNT002  ; 第一步时间
ANDNOT 26.01  ; 第2步时间为0
MOV(21) CNT3 DM935  ; 步序时间显示
; rung 65
LD CNT003  ; 第二步时间
ANDNOT 26.02  ; 第3步时间为0
MOV(21) CNT4 DM935  ; 步序时间显示
; rung 66
LD CNT004  ; 第三步时间
ANDNOT 26.03  ; 第4步时间为0
MOV(21) CNT5 DM935  ; 步序时间显示
; rung 67
LD CNT005  ; 第4步时间
ANDNOT 26.04  ; 第5步时间为0
MOV(21) CNT6 DM935  ; 步序时间显示
; rung 68
LD CNT006  ; 第五步时间
ANDNOT 26.05  ; 第6步时间为0
MOV(21) CNT7 DM935  ; 步序时间显示

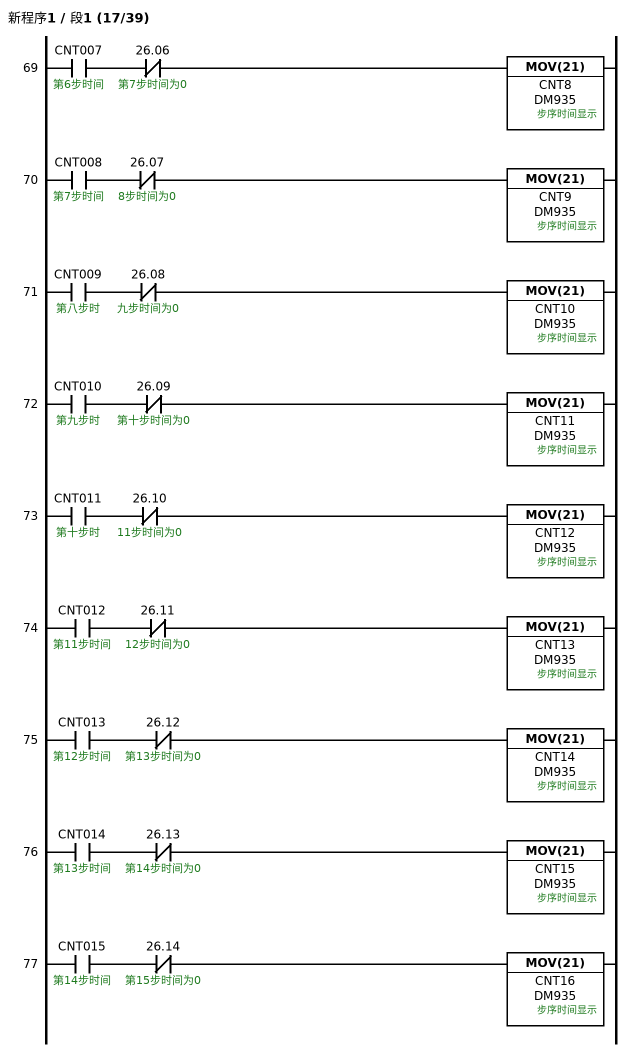
; rung 69
LD CNT007  ; 第6步时间
ANDNOT 26.06  ; 第7步时间为0
MOV(21) CNT8 DM935  ; 步序时间显示
; rung 70
LD CNT008  ; 第7步时间
ANDNOT 26.07  ; 8步时间为0
MOV(21) CNT9 DM935  ; 步序时间显示
; rung 71
LD CNT009  ; 第八步时
ANDNOT 26.08  ; 九步时间为0
MOV(21) CNT10 DM935  ; 步序时间显示
; rung 72
LD CNT010  ; 第九步时
ANDNOT 26.09  ; 第十步时间为0
MOV(21) CNT11 DM935  ; 步序时间显示
; rung 73
LD CNT011  ; 第十步时
ANDNOT 26.10  ; 11步时间为0
MOV(21) CNT12 DM935  ; 步序时间显示
; rung 74
LD CNT012  ; 第11步时间
ANDNOT 26.11  ; 12步时间为0
MOV(21) CNT13 DM935  ; 步序时间显示
; rung 75
LD CNT013  ; 第12步时间
ANDNOT 26.12  ; 第13步时间为0
MOV(21) CNT14 DM935  ; 步序时间显示
; rung 76
LD CNT014  ; 第13步时间
ANDNOT 26.13  ; 第14步时间为0
MOV(21) CNT15 DM935  ; 步序时间显示
; rung 77
LD CNT015  ; 第14步时间
ANDNOT 26.14  ; 第15步时间为0
MOV(21) CNT16 DM935  ; 步序时间显示

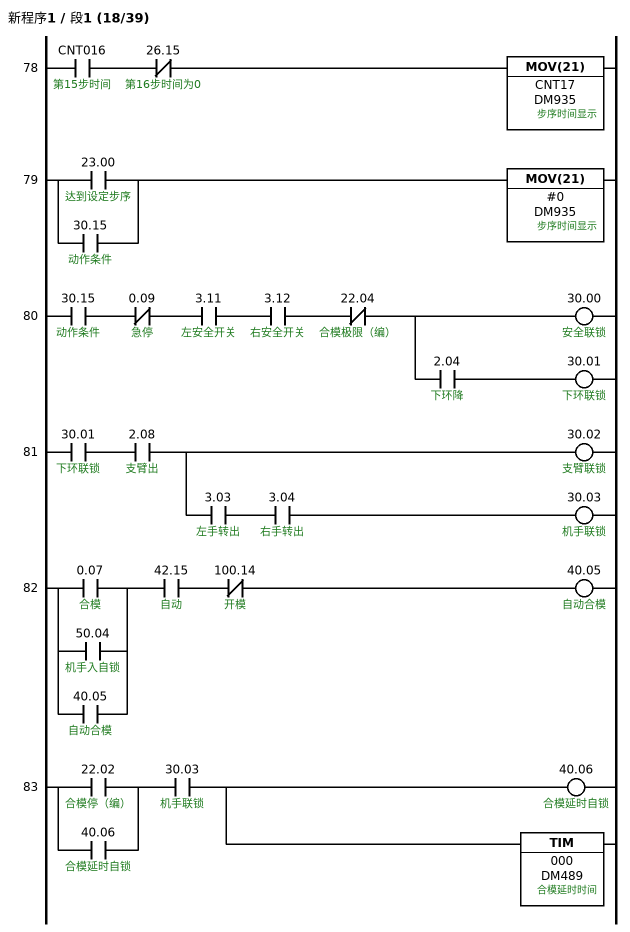
; rung 78
LD CNT016  ; 第15步时间
ANDNOT 26.15  ; 第16步时间为0
MOV(21) CNT17 DM935  ; 步序时间显示
; rung 79
LD 23.00  ; 达到设定步序
OR 30.15  ; 动作条件
MOV(21) #0 DM935  ; 步序时间显示
; rung 80
LD 30.15  ; 动作条件
ANDNOT 0.09  ; 急停
AND 3.11  ; 左安全开关
AND 3.12  ; 右安全开关
ANDNOT 22.04  ; 合模极限（编）
OUT 30.00  ; 安全联锁
AND 2.04  ; 下环降
OUT 30.01  ; 下环联锁
; rung 81
LD 30.01  ; 下环联锁
AND 2.08  ; 支臂出
OUT 30.02  ; 支臂联锁
AND 3.03  ; 左手转出
AND 3.04  ; 右手转出
OUT 30.03  ; 机手联锁
; rung 82
LD 0.07  ; 合模
OR 50.04  ; 机手入自锁
OR 40.05  ; 自动合模
AND 42.15  ; 自动
ANDNOT 100.14  ; 开模
OUT 40.05  ; 自动合模
; rung 83
LD 22.02  ; 合模停（编）
OR 40.06  ; 合模延时自锁
AND 30.03  ; 机手联锁
OUT 40.06  ; 合模延时自锁
TIM 000 DM489  ; 合模延时时间

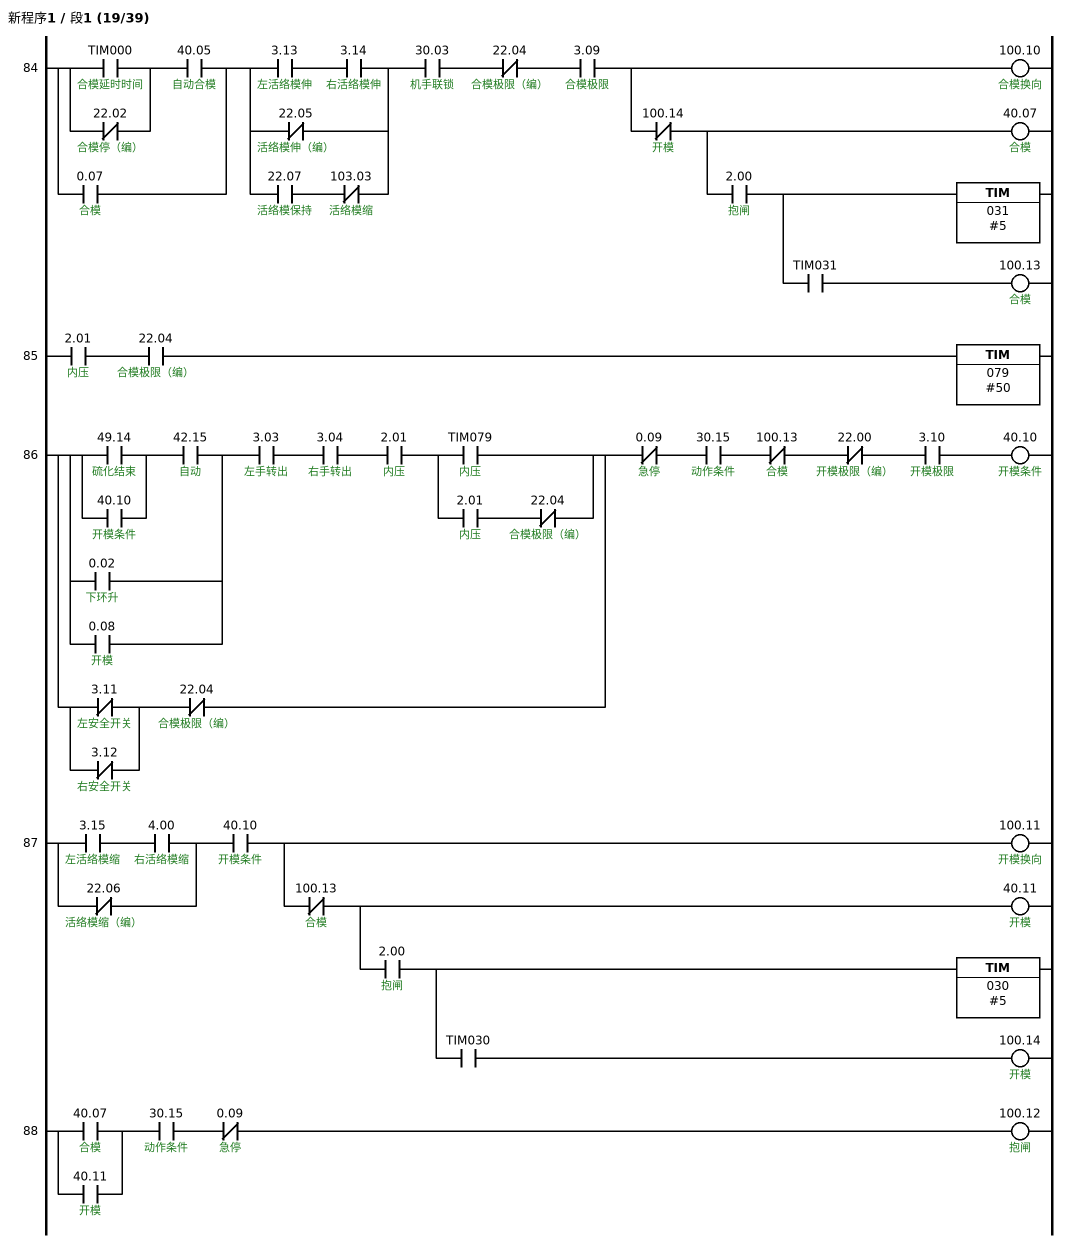
; rung 84
LD TIM000  ; 合模延时时间
ORNOT 22.02  ; 合模停（编）
AND 40.05  ; 自动合模
OR 0.07  ; 合模
LD 3.13  ; 左活络模伸
AND 3.14  ; 右活络模伸
ORNOT 22.05  ; 活络模伸（编）
LD 22.07  ; 活络模保持
ANDNOT 103.03  ; 活络模缩
ORLD
ANDLD
AND 30.03  ; 机手联锁
ANDNOT 22.04  ; 合模极限（编）
AND 3.09  ; 合模极限
OUT 100.10  ; 合模换向
ANDNOT 100.14  ; 开模
OUT 40.07  ; 合模
AND 2.00  ; 抱闸
TIM 031 #5
AND TIM031
OUT 100.13  ; 合模
; rung 85
LD 2.01  ; 内压
AND 22.04  ; 合模极限（编）
TIM 079 #50
; rung 86
LD 49.14  ; 硫化结束
OR 40.10  ; 开模条件
AND 42.15  ; 自动
OR 0.02  ; 下环升
OR 0.08  ; 开模
AND 3.03  ; 左手转出
AND 3.04  ; 右手转出
AND 2.01  ; 内压
LD TIM079  ; 内压
LD 2.01  ; 内压
ANDNOT 22.04  ; 合模极限（编）
ORLD
ANDLD
LDNOT 3.11  ; 左安全开关
ORNOT 3.12  ; 右安全开关
ANDNOT 22.04  ; 合模极限（编）
ORLD
ANDNOT 0.09  ; 急停
AND 30.15  ; 动作条件
ANDNOT 100.13  ; 合模
ANDNOT 22.00  ; 开模极限（编）
AND 3.10  ; 开模极限
OUT 40.10  ; 开模条件
; rung 87
LD 3.15  ; 左活络模缩
AND 4.00  ; 右活络模缩
ORNOT 22.06  ; 活络模缩（编）
AND 40.10  ; 开模条件
OUT 100.11  ; 开模换向
ANDNOT 100.13  ; 合模
OUT 40.11  ; 开模
AND 2.00  ; 抱闸
TIM 030 #5
AND TIM030
OUT 100.14  ; 开模
; rung 88
LD 40.07  ; 合模
OR 40.11  ; 开模
AND 30.15  ; 动作条件
ANDNOT 0.09  ; 急停
OUT 100.12  ; 抱闸

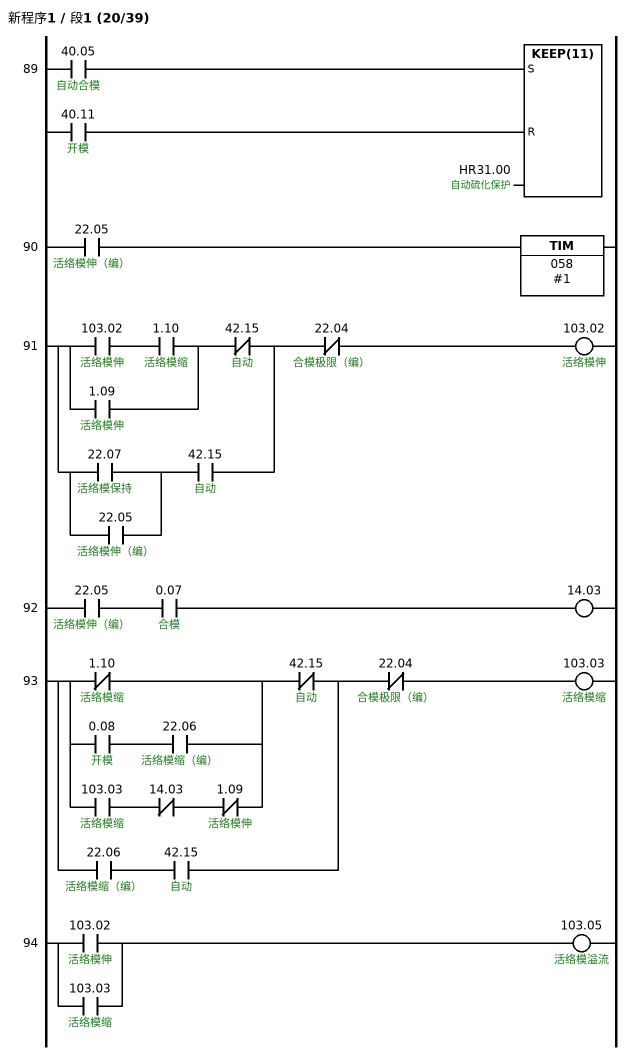
; rung 89
LD 40.05  ; 自动合模
LD 40.11  ; 开模
KEEP(11) HR31.00  ; 自动硫化保护
; rung 90
LD 22.05  ; 活络模伸（编）
TIM 058 #1
; rung 91
LD 103.02  ; 活络模伸
AND 1.10  ; 活络模缩
OR 1.09  ; 活络模伸
ANDNOT 42.15  ; 自动
LD 22.07  ; 活络模保持
OR 22.05  ; 活络模伸（编）
AND 42.15  ; 自动
ORLD
ANDNOT 22.04  ; 合模极限（编）
OUT 103.02  ; 活络模伸
; rung 92
LD 22.05  ; 活络模伸（编）
AND 0.07  ; 合模
OUT 14.03
; rung 93
LDNOT 1.10  ; 活络模缩
LD 0.08  ; 开模
AND 22.06  ; 活络模缩（编）
ORLD
LD 103.03  ; 活络模缩
ANDNOT 14.03
ANDNOT 1.09  ; 活络模伸
ORLD
ANDNOT 42.15  ; 自动
LD 22.06  ; 活络模缩（编）
AND 42.15  ; 自动
ORLD
ANDNOT 22.04  ; 合模极限（编）
OUT 103.03  ; 活络模缩
; rung 94
LD 103.02  ; 活络模伸
OR 103.03  ; 活络模缩
OUT 103.05  ; 活络模溢流

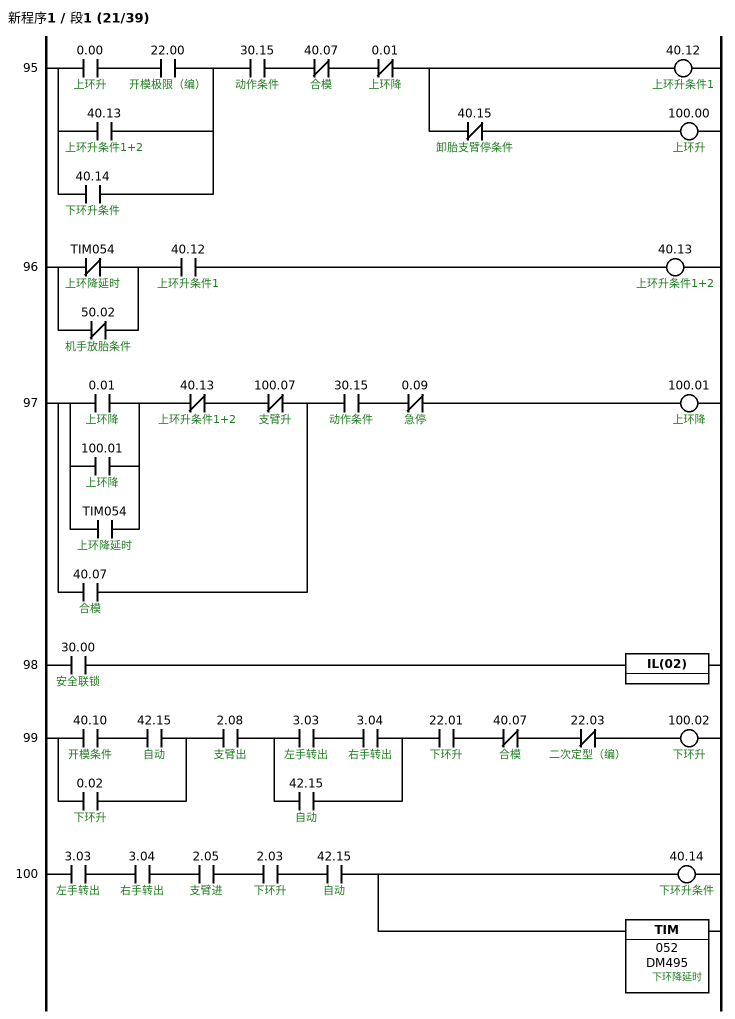
; rung 95
LD 0.00  ; 上环升
AND 22.00  ; 开模极限（编）
OR 40.13  ; 上环升条件1+2
OR 40.14  ; 下环升条件
AND 30.15  ; 动作条件
ANDNOT 40.07  ; 合模
ANDNOT 0.01  ; 上环降
OUT 40.12  ; 上环升条件1
ANDNOT 40.15  ; 卸胎支臂停条件
OUT 100.00  ; 上环升
; rung 96
LDNOT TIM054  ; 上环降延时
ORNOT 50.02  ; 机手放胎条件
AND 40.12  ; 上环升条件1
OUT 40.13  ; 上环升条件1+2
; rung 97
LD 0.01  ; 上环降
OR 100.01  ; 上环降
OR TIM054  ; 上环降延时
ANDNOT 40.13  ; 上环升条件1+2
ANDNOT 100.07  ; 支臂升
OR 40.07  ; 合模
AND 30.15  ; 动作条件
ANDNOT 0.09  ; 急停
OUT 100.01  ; 上环降
; rung 98
LD 30.00  ; 安全联锁
IL(02)
; rung 99
LD 40.10  ; 开模条件
AND 42.15  ; 自动
OR 0.02  ; 下环升
AND 2.08  ; 支臂出
LD 3.03  ; 左手转出
AND 3.04  ; 右手转出
OR 42.15  ; 自动
ANDLD
AND 22.01  ; 下环升
ANDNOT 40.07  ; 合模
ANDNOT 22.03  ; 二次定型（编）
OUT 100.02  ; 下环升
; rung 100
LD 3.03  ; 左手转出
AND 3.04  ; 右手转出
AND 2.05  ; 支臂进
AND 2.03  ; 下环升
AND 42.15  ; 自动
OUT 40.14  ; 下环升条件
TIM 052 DM495  ; 下环降延时

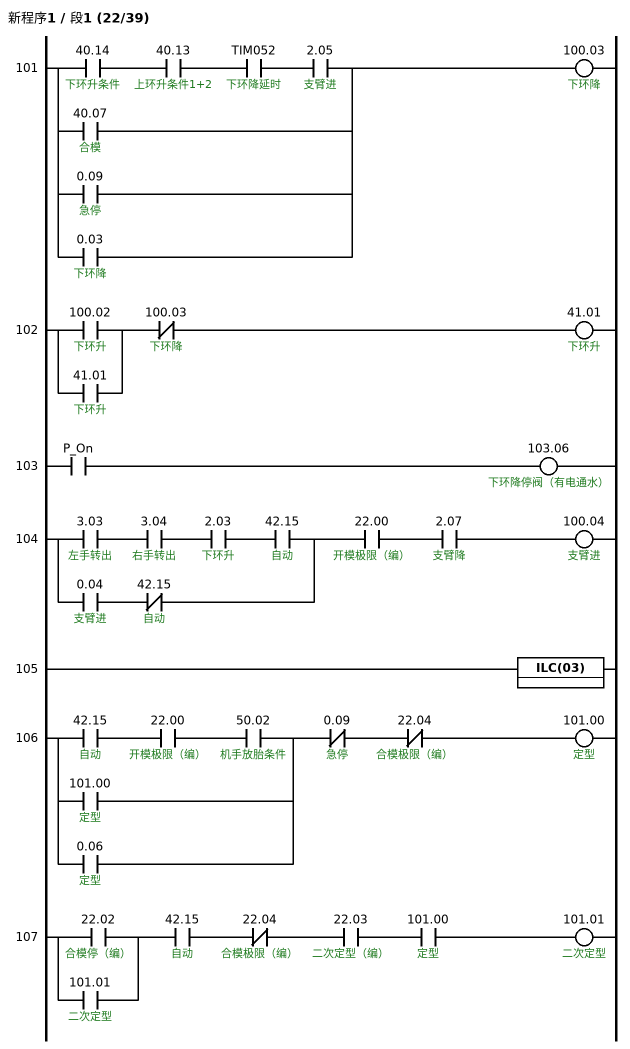
; rung 101
LD 40.14  ; 下环升条件
AND 40.13  ; 上环升条件1+2
AND TIM052  ; 下环降延时
AND 2.05  ; 支臂进
OR 40.07  ; 合模
OR 0.09  ; 急停
OR 0.03  ; 下环降
OUT 100.03  ; 下环降
; rung 102
LD 100.02  ; 下环升
OR 41.01  ; 下环升
ANDNOT 100.03  ; 下环降
OUT 41.01  ; 下环升
; rung 103
LD P_On
OUT 103.06  ; 下环降停阀（有电通水）
; rung 104
LD 3.03  ; 左手转出
AND 3.04  ; 右手转出
AND 2.03  ; 下环升
AND 42.15  ; 自动
LD 0.04  ; 支臂进
ANDNOT 42.15  ; 自动
ORLD
AND 22.00  ; 开模极限（编）
AND 2.07  ; 支臂降
OUT 100.04  ; 支臂进
; rung 105
ILC(03)
; rung 106
LD 42.15  ; 自动
AND 22.00  ; 开模极限（编）
AND 50.02  ; 机手放胎条件
OR 101.00  ; 定型
OR 0.06  ; 定型
ANDNOT 0.09  ; 急停
ANDNOT 22.04  ; 合模极限（编）
OUT 101.00  ; 定型
; rung 107
LD 22.02  ; 合模停（编）
OR 101.01  ; 二次定型
AND 42.15  ; 自动
ANDNOT 22.04  ; 合模极限（编）
AND 22.03  ; 二次定型（编）
AND 101.00  ; 定型
OUT 101.01  ; 二次定型

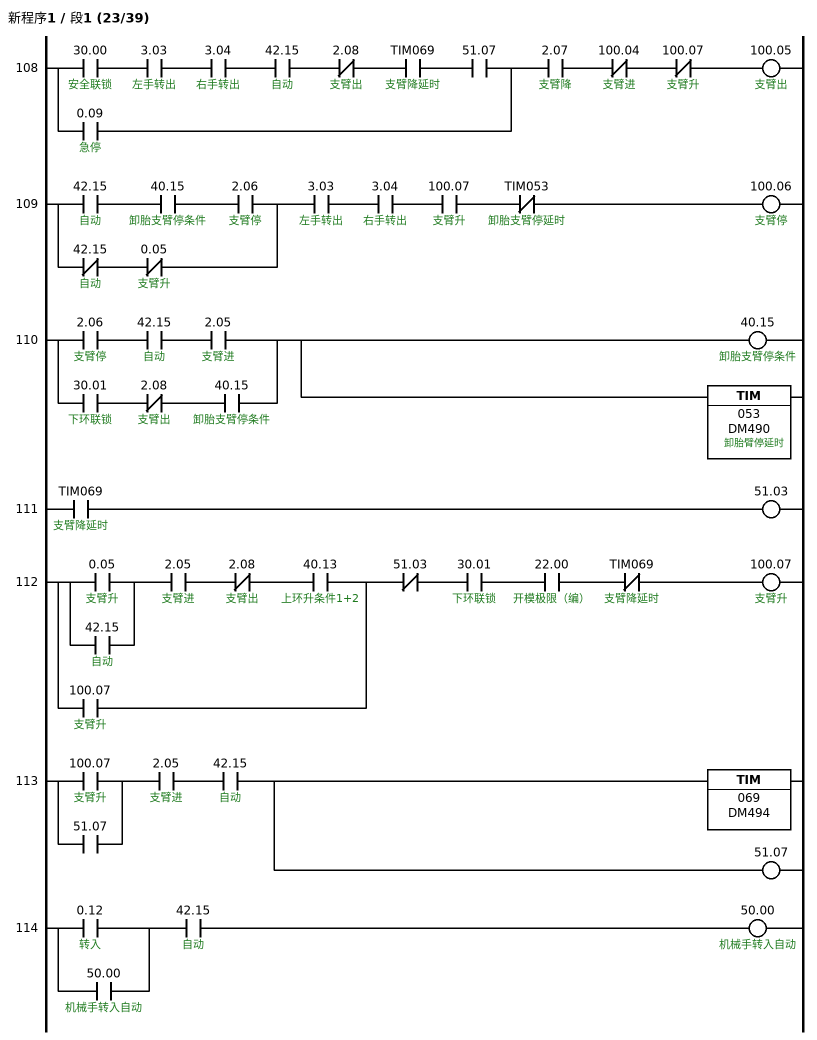
; rung 108
LD 30.00  ; 安全联锁
AND 3.03  ; 左手转出
AND 3.04  ; 右手转出
AND 42.15  ; 自动
ANDNOT 2.08  ; 支臂出
AND TIM069  ; 支臂降延时
AND 51.07
OR 0.09  ; 急停
AND 2.07  ; 支臂降
ANDNOT 100.04  ; 支臂进
ANDNOT 100.07  ; 支臂升
OUT 100.05  ; 支臂出
; rung 109
LD 42.15  ; 自动
AND 40.15  ; 卸胎支臂停条件
AND 2.06  ; 支臂停
LDNOT 42.15  ; 自动
ANDNOT 0.05  ; 支臂升
ORLD
AND 3.03  ; 左手转出
AND 3.04  ; 右手转出
AND 100.07  ; 支臂升
ANDNOT TIM053  ; 卸胎支臂停延时
OUT 100.06  ; 支臂停
; rung 110
LD 2.06  ; 支臂停
AND 42.15  ; 自动
AND 2.05  ; 支臂进
LD 30.01  ; 下环联锁
ANDNOT 2.08  ; 支臂出
AND 40.15  ; 卸胎支臂停条件
ORLD
OUT 40.15  ; 卸胎支臂停条件
TIM 053 DM490  ; 卸胎臂停延时
; rung 111
LD TIM069  ; 支臂降延时
OUT 51.03
; rung 112
LD 0.05  ; 支臂升
OR 42.15  ; 自动
AND 2.05  ; 支臂进
ANDNOT 2.08  ; 支臂出
AND 40.13  ; 上环升条件1+2
OR 100.07  ; 支臂升
ANDNOT 51.03
AND 30.01  ; 下环联锁
AND 22.00  ; 开模极限（编）
ANDNOT TIM069  ; 支臂降延时
OUT 100.07  ; 支臂升
; rung 113
LD 100.07  ; 支臂升
OR 51.07
AND 2.05  ; 支臂进
AND 42.15  ; 自动
TIM 069 DM494
OUT 51.07
; rung 114
LD 0.12  ; 转入
OR 50.00  ; 机械手转入自动
AND 42.15  ; 自动
OUT 50.00  ; 机械手转入自动

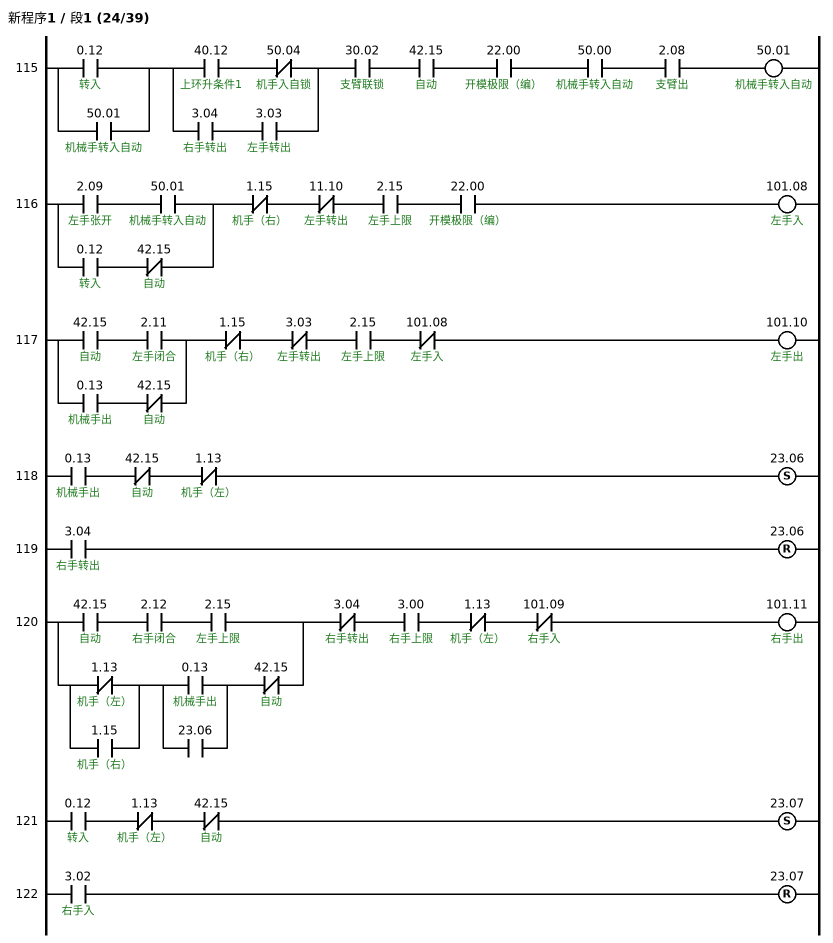
; rung 115
LD 0.12  ; 转入
OR 50.01  ; 机械手转入自动
LD 40.12  ; 上环升条件1
ANDNOT 50.04  ; 机手入自锁
LD 3.04  ; 右手转出
AND 3.03  ; 左手转出
ORLD
ANDLD
AND 30.02  ; 支臂联锁
AND 42.15  ; 自动
AND 22.00  ; 开模极限（编）
AND 50.00  ; 机械手转入自动
AND 2.08  ; 支臂出
OUT 50.01  ; 机械手转入自动
; rung 116
LD 2.09  ; 左手张开
AND 50.01  ; 机械手转入自动
LD 0.12  ; 转入
ANDNOT 42.15  ; 自动
ORLD
ANDNOT 1.15  ; 机手（右）
ANDNOT 11.10  ; 左手转出
AND 2.15  ; 左手上限
AND 22.00  ; 开模极限（编）
OUT 101.08  ; 左手入
; rung 117
LD 42.15  ; 自动
AND 2.11  ; 左手闭合
LD 0.13  ; 机械手出
ANDNOT 42.15  ; 自动
ORLD
ANDNOT 1.15  ; 机手（右）
ANDNOT 3.03  ; 左手转出
AND 2.15  ; 左手上限
ANDNOT 101.08  ; 左手入
OUT 101.10  ; 左手出
; rung 118
LD 0.13  ; 机械手出
ANDNOT 42.15  ; 自动
ANDNOT 1.13  ; 机手（左）
SET 23.06
; rung 119
LD 3.04  ; 右手转出
RSET 23.06
; rung 120
LD 42.15  ; 自动
AND 2.12  ; 右手闭合
AND 2.15  ; 左手上限
LDNOT 1.13  ; 机手（左）
OR 1.15  ; 机手（右）
LD 0.13  ; 机械手出
OR 23.06
ANDLD
ANDNOT 42.15  ; 自动
ORLD
ANDNOT 3.04  ; 右手转出
AND 3.00  ; 右手上限
ANDNOT 1.13  ; 机手（左）
ANDNOT 101.09  ; 右手入
OUT 101.11  ; 右手出
; rung 121
LD 0.12  ; 转入
ANDNOT 1.13  ; 机手（左）
ANDNOT 42.15  ; 自动
SET 23.07
; rung 122
LD 3.02  ; 右手入
RSET 23.07

